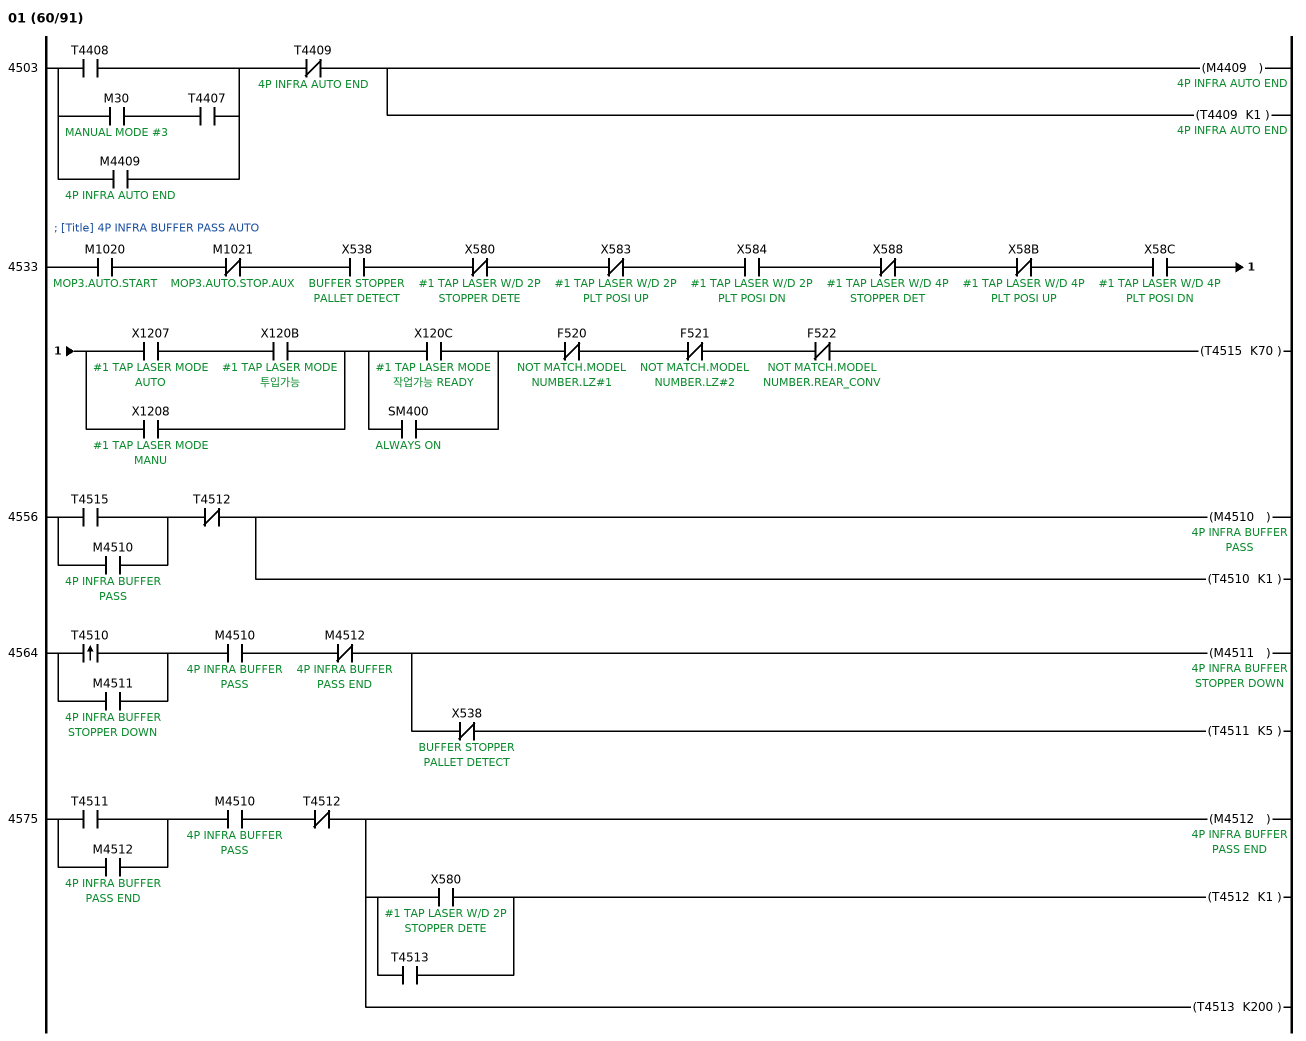
4503  LD      T4408
      LD      M30  ; MANUAL MODE #3
      AND     T4407
      ORB
      OR      M4409  ; 4P INFRA AUTO END
      ANI     T4409  ; 4P INFRA AUTO END
      OUT     M4409  ; 4P INFRA AUTO END
      OUT     T4409 K1  ; 4P INFRA AUTO END
; [Title] 4P INFRA BUFFER PASS AUTO
4533  LD      M1020  ; MOP3.AUTO.START
      ANI     M1021  ; MOP3.AUTO.STOP.AUX
      AND     X538  ; BUFFER STOPPER PALLET DETECT
      ANI     X580  ; #1 TAP LASER W/D 2P STOPPER DETE
      ANI     X583  ; #1 TAP LASER W/D 2P PLT POSI UP
      AND     X584  ; #1 TAP LASER W/D 2P PLT POSI DN
      ANI     X588  ; #1 TAP LASER W/D 4P STOPPER DET
      ANI     X58B  ; #1 TAP LASER W/D 4P PLT POSI UP
      AND     X58C  ; #1 TAP LASER W/D 4P PLT POSI DN
      LD      X1207  ; #1 TAP LASER MODE AUTO
      AND     X120B  ; #1 TAP LASER MODE 투입가능
      OR      X1208  ; #1 TAP LASER MODE MANU
      ANB
      LD      X120C  ; #1 TAP LASER MODE 작업가능 READY
      OR      SM400  ; ALWAYS ON
      ANB
      ANI     F520  ; NOT MATCH.MODEL NUMBER.LZ#1
      ANI     F521  ; NOT MATCH.MODEL NUMBER.LZ#2
      ANI     F522  ; NOT MATCH.MODEL NUMBER.REAR_CONV
      OUT     T4515 K70
4556  LD      T4515
      OR      M4510  ; 4P INFRA BUFFER PASS
      ANI     T4512
      OUT     M4510  ; 4P INFRA BUFFER PASS
      OUT     T4510 K1
4564  LDP     T4510
      OR      M4511  ; 4P INFRA BUFFER STOPPER DOWN
      AND     M4510  ; 4P INFRA BUFFER PASS
      ANI     M4512  ; 4P INFRA BUFFER PASS END
      OUT     M4511  ; 4P INFRA BUFFER STOPPER DOWN
      ANI     X538  ; BUFFER STOPPER PALLET DETECT
      OUT     T4511 K5
4575  LD      T4511
      OR      M4512  ; 4P INFRA BUFFER PASS END
      AND     M4510  ; 4P INFRA BUFFER PASS
      ANI     T4512
      OUT     M4512  ; 4P INFRA BUFFER PASS END
      MPS
      LD      X580  ; #1 TAP LASER W/D 2P STOPPER DETE
      OR      T4513
      ANB
      OUT     T4512 K1
      MPP
      OUT     T4513 K200
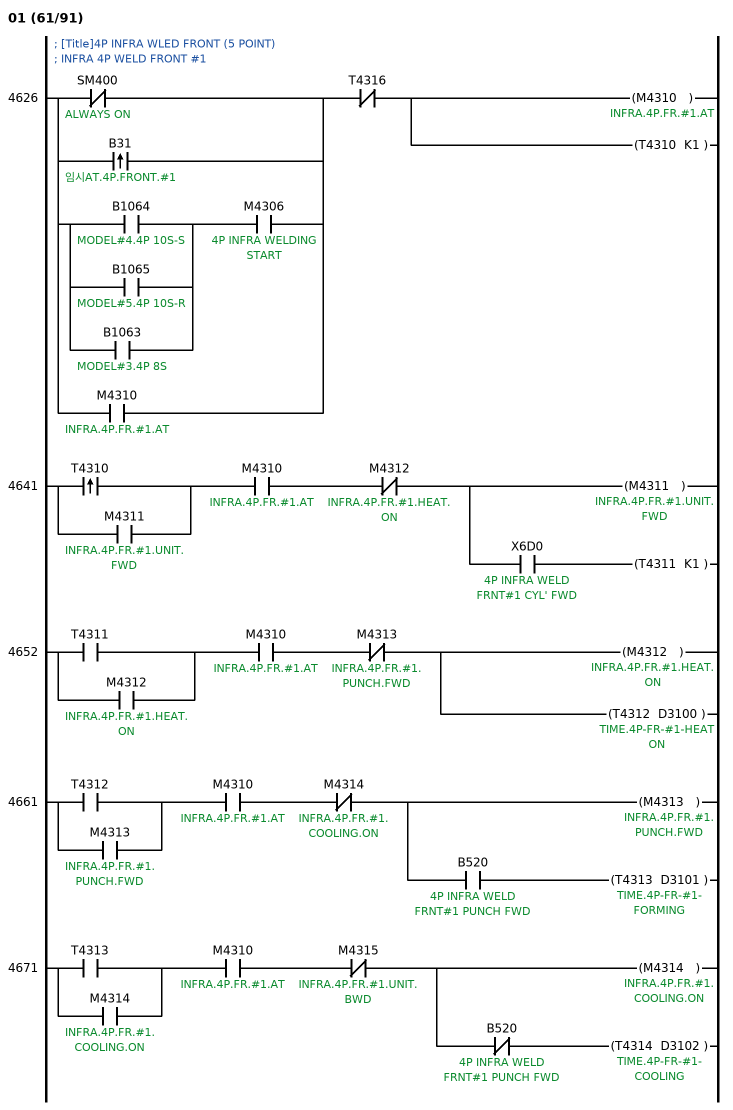
; [Title]4P INFRA WLED FRONT (5 POINT)
; INFRA 4P WELD FRONT #1
4626  LDI     SM400  ; ALWAYS ON
      ORP     B31  ; 임시AT.4P.FRONT.#1
      LD      B1064  ; MODEL#4.4P 10S-S
      OR      B1065  ; MODEL#5.4P 10S-R
      OR      B1063  ; MODEL#3.4P 8S
      AND     M4306  ; 4P INFRA WELDING START
      ORB
      OR      M4310  ; INFRA.4P.FR.#1.AT
      ANI     T4316
      OUT     M4310  ; INFRA.4P.FR.#1.AT
      OUT     T4310 K1
4641  LDP     T4310
      OR      M4311  ; INFRA.4P.FR.#1.UNIT.FWD
      AND     M4310  ; INFRA.4P.FR.#1.AT
      ANI     M4312  ; INFRA.4P.FR.#1.HEAT.ON
      OUT     M4311  ; INFRA.4P.FR.#1.UNIT.FWD
      AND     X6D0  ; 4P INFRA WELD FRNT#1 CYL' FWD
      OUT     T4311 K1
4652  LD      T4311
      OR      M4312  ; INFRA.4P.FR.#1.HEAT.ON
      AND     M4310  ; INFRA.4P.FR.#1.AT
      ANI     M4313  ; INFRA.4P.FR.#1.PUNCH.FWD
      OUT     M4312  ; INFRA.4P.FR.#1.HEAT.ON
      OUT     T4312 D3100  ; TIME.4P-FR-#1-HEAT ON
4661  LD      T4312
      OR      M4313  ; INFRA.4P.FR.#1.PUNCH.FWD
      AND     M4310  ; INFRA.4P.FR.#1.AT
      ANI     M4314  ; INFRA.4P.FR.#1.COOLING.ON
      OUT     M4313  ; INFRA.4P.FR.#1.PUNCH.FWD
      AND     B520  ; 4P INFRA WELD FRNT#1 PUNCH FWD
      OUT     T4313 D3101  ; TIME.4P-FR-#1-FORMING
4671  LD      T4313
      OR      M4314  ; INFRA.4P.FR.#1.COOLING.ON
      AND     M4310  ; INFRA.4P.FR.#1.AT
      ANI     M4315  ; INFRA.4P.FR.#1.UNIT.BWD
      OUT     M4314  ; INFRA.4P.FR.#1.COOLING.ON
      ANI     B520  ; 4P INFRA WELD FRNT#1 PUNCH FWD
      OUT     T4314 D3102  ; TIME.4P-FR-#1-COOLING
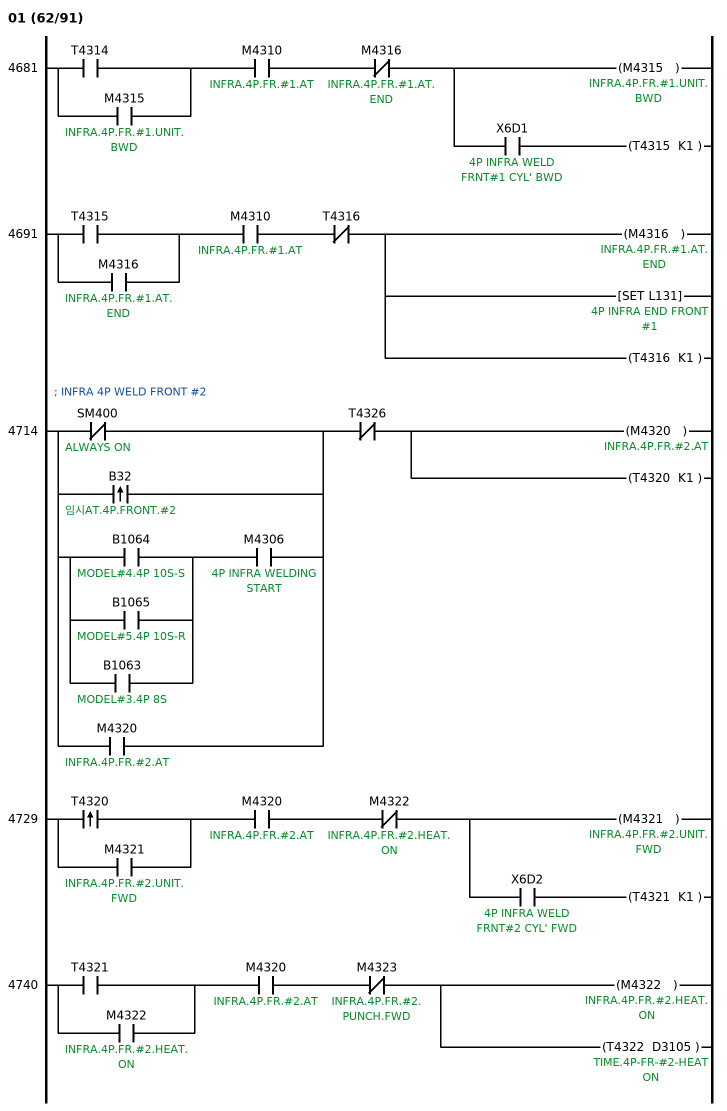
4681  LD      T4314
      OR      M4315  ; INFRA.4P.FR.#1.UNIT.BWD
      AND     M4310  ; INFRA.4P.FR.#1.AT
      ANI     M4316  ; INFRA.4P.FR.#1.AT.END
      OUT     M4315  ; INFRA.4P.FR.#1.UNIT.BWD
      AND     X6D1  ; 4P INFRA WELD FRNT#1 CYL' BWD
      OUT     T4315 K1
4691  LD      T4315
      OR      M4316  ; INFRA.4P.FR.#1.AT.END
      AND     M4310  ; INFRA.4P.FR.#1.AT
      ANI     T4316
      OUT     M4316  ; INFRA.4P.FR.#1.AT.END
      SET     L131  ; 4P INFRA END FRONT #1
      OUT     T4316 K1
; INFRA 4P WELD FRONT #2
4714  LDI     SM400  ; ALWAYS ON
      ORP     B32  ; 임시AT.4P.FRONT.#2
      LD      B1064  ; MODEL#4.4P 10S-S
      OR      B1065  ; MODEL#5.4P 10S-R
      OR      B1063  ; MODEL#3.4P 8S
      AND     M4306  ; 4P INFRA WELDING START
      ORB
      OR      M4320  ; INFRA.4P.FR.#2.AT
      ANI     T4326
      OUT     M4320  ; INFRA.4P.FR.#2.AT
      OUT     T4320 K1
4729  LDP     T4320
      OR      M4321  ; INFRA.4P.FR.#2.UNIT.FWD
      AND     M4320  ; INFRA.4P.FR.#2.AT
      ANI     M4322  ; INFRA.4P.FR.#2.HEAT.ON
      OUT     M4321  ; INFRA.4P.FR.#2.UNIT.FWD
      AND     X6D2  ; 4P INFRA WELD FRNT#2 CYL' FWD
      OUT     T4321 K1
4740  LD      T4321
      OR      M4322  ; INFRA.4P.FR.#2.HEAT.ON
      AND     M4320  ; INFRA.4P.FR.#2.AT
      ANI     M4323  ; INFRA.4P.FR.#2.PUNCH.FWD
      OUT     M4322  ; INFRA.4P.FR.#2.HEAT.ON
      OUT     T4322 D3105  ; TIME.4P-FR-#2-HEAT ON
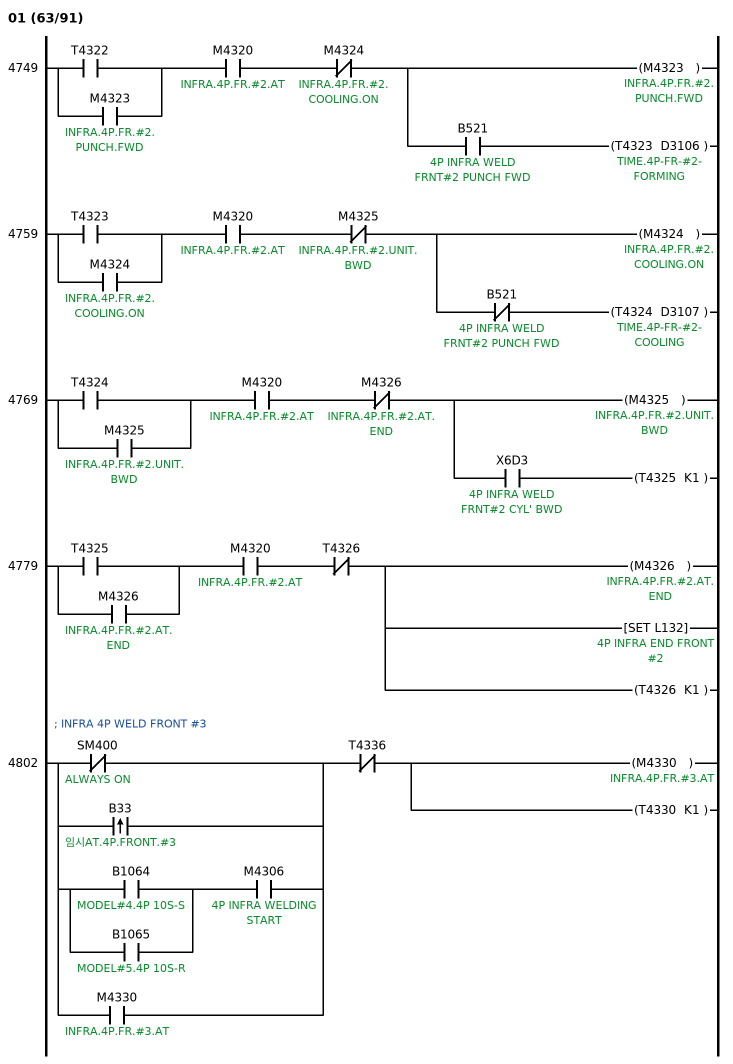
4749  LD      T4322
      OR      M4323  ; INFRA.4P.FR.#2.PUNCH.FWD
      AND     M4320  ; INFRA.4P.FR.#2.AT
      ANI     M4324  ; INFRA.4P.FR.#2.COOLING.ON
      OUT     M4323  ; INFRA.4P.FR.#2.PUNCH.FWD
      AND     B521  ; 4P INFRA WELD FRNT#2 PUNCH FWD
      OUT     T4323 D3106  ; TIME.4P-FR-#2-FORMING
4759  LD      T4323
      OR      M4324  ; INFRA.4P.FR.#2.COOLING.ON
      AND     M4320  ; INFRA.4P.FR.#2.AT
      ANI     M4325  ; INFRA.4P.FR.#2.UNIT.BWD
      OUT     M4324  ; INFRA.4P.FR.#2.COOLING.ON
      ANI     B521  ; 4P INFRA WELD FRNT#2 PUNCH FWD
      OUT     T4324 D3107  ; TIME.4P-FR-#2-COOLING
4769  LD      T4324
      OR      M4325  ; INFRA.4P.FR.#2.UNIT.BWD
      AND     M4320  ; INFRA.4P.FR.#2.AT
      ANI     M4326  ; INFRA.4P.FR.#2.AT.END
      OUT     M4325  ; INFRA.4P.FR.#2.UNIT.BWD
      AND     X6D3  ; 4P INFRA WELD FRNT#2 CYL' BWD
      OUT     T4325 K1
4779  LD      T4325
      OR      M4326  ; INFRA.4P.FR.#2.AT.END
      AND     M4320  ; INFRA.4P.FR.#2.AT
      ANI     T4326
      OUT     M4326  ; INFRA.4P.FR.#2.AT.END
      SET     L132  ; 4P INFRA END FRONT #2
      OUT     T4326 K1
; INFRA 4P WELD FRONT #3
4802  LDI     SM400  ; ALWAYS ON
      ORP     B33  ; 임시AT.4P.FRONT.#3
      LD      B1064  ; MODEL#4.4P 10S-S
      OR      B1065  ; MODEL#5.4P 10S-R
      AND     M4306  ; 4P INFRA WELDING START
      ORB
      OR      M4330  ; INFRA.4P.FR.#3.AT
      ANI     T4336
      OUT     M4330  ; INFRA.4P.FR.#3.AT
      OUT     T4330 K1
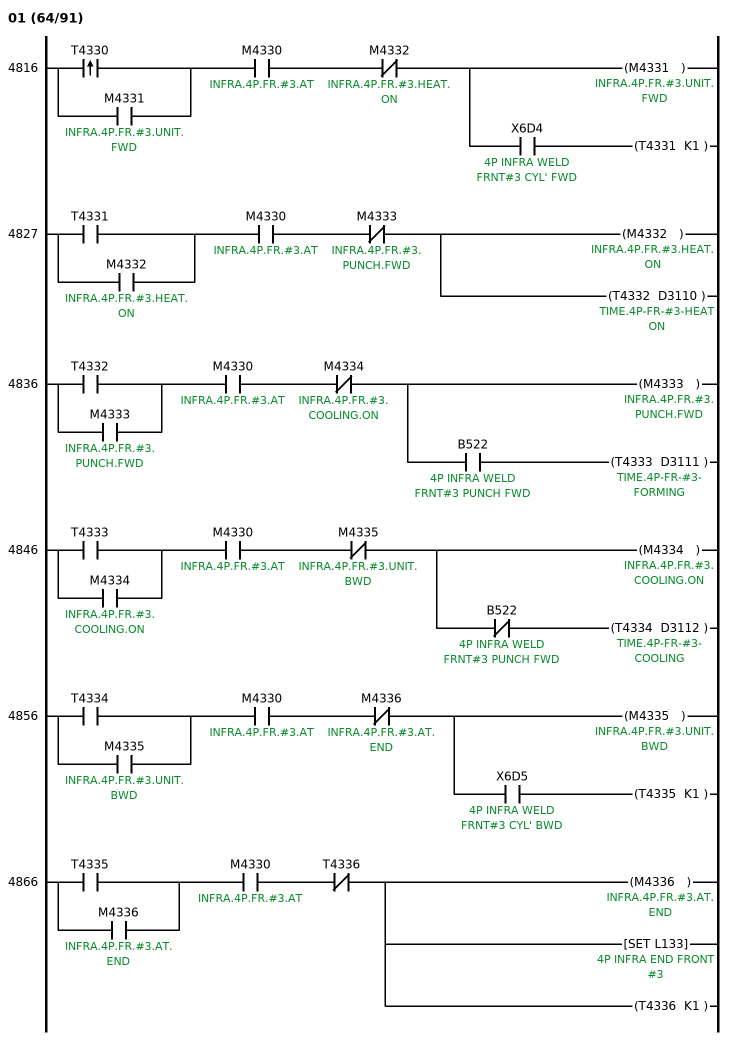
4816  LDP     T4330
      OR      M4331  ; INFRA.4P.FR.#3.UNIT.FWD
      AND     M4330  ; INFRA.4P.FR.#3.AT
      ANI     M4332  ; INFRA.4P.FR.#3.HEAT.ON
      OUT     M4331  ; INFRA.4P.FR.#3.UNIT.FWD
      AND     X6D4  ; 4P INFRA WELD FRNT#3 CYL' FWD
      OUT     T4331 K1
4827  LD      T4331
      OR      M4332  ; INFRA.4P.FR.#3.HEAT.ON
      AND     M4330  ; INFRA.4P.FR.#3.AT
      ANI     M4333  ; INFRA.4P.FR.#3.PUNCH.FWD
      OUT     M4332  ; INFRA.4P.FR.#3.HEAT.ON
      OUT     T4332 D3110  ; TIME.4P-FR-#3-HEAT ON
4836  LD      T4332
      OR      M4333  ; INFRA.4P.FR.#3.PUNCH.FWD
      AND     M4330  ; INFRA.4P.FR.#3.AT
      ANI     M4334  ; INFRA.4P.FR.#3.COOLING.ON
      OUT     M4333  ; INFRA.4P.FR.#3.PUNCH.FWD
      AND     B522  ; 4P INFRA WELD FRNT#3 PUNCH FWD
      OUT     T4333 D3111  ; TIME.4P-FR-#3-FORMING
4846  LD      T4333
      OR      M4334  ; INFRA.4P.FR.#3.COOLING.ON
      AND     M4330  ; INFRA.4P.FR.#3.AT
      ANI     M4335  ; INFRA.4P.FR.#3.UNIT.BWD
      OUT     M4334  ; INFRA.4P.FR.#3.COOLING.ON
      ANI     B522  ; 4P INFRA WELD FRNT#3 PUNCH FWD
      OUT     T4334 D3112  ; TIME.4P-FR-#3-COOLING
4856  LD      T4334
      OR      M4335  ; INFRA.4P.FR.#3.UNIT.BWD
      AND     M4330  ; INFRA.4P.FR.#3.AT
      ANI     M4336  ; INFRA.4P.FR.#3.AT.END
      OUT     M4335  ; INFRA.4P.FR.#3.UNIT.BWD
      AND     X6D5  ; 4P INFRA WELD FRNT#3 CYL' BWD
      OUT     T4335 K1
4866  LD      T4335
      OR      M4336  ; INFRA.4P.FR.#3.AT.END
      AND     M4330  ; INFRA.4P.FR.#3.AT
      ANI     T4336
      OUT     M4336  ; INFRA.4P.FR.#3.AT.END
      SET     L133  ; 4P INFRA END FRONT #3
      OUT     T4336 K1
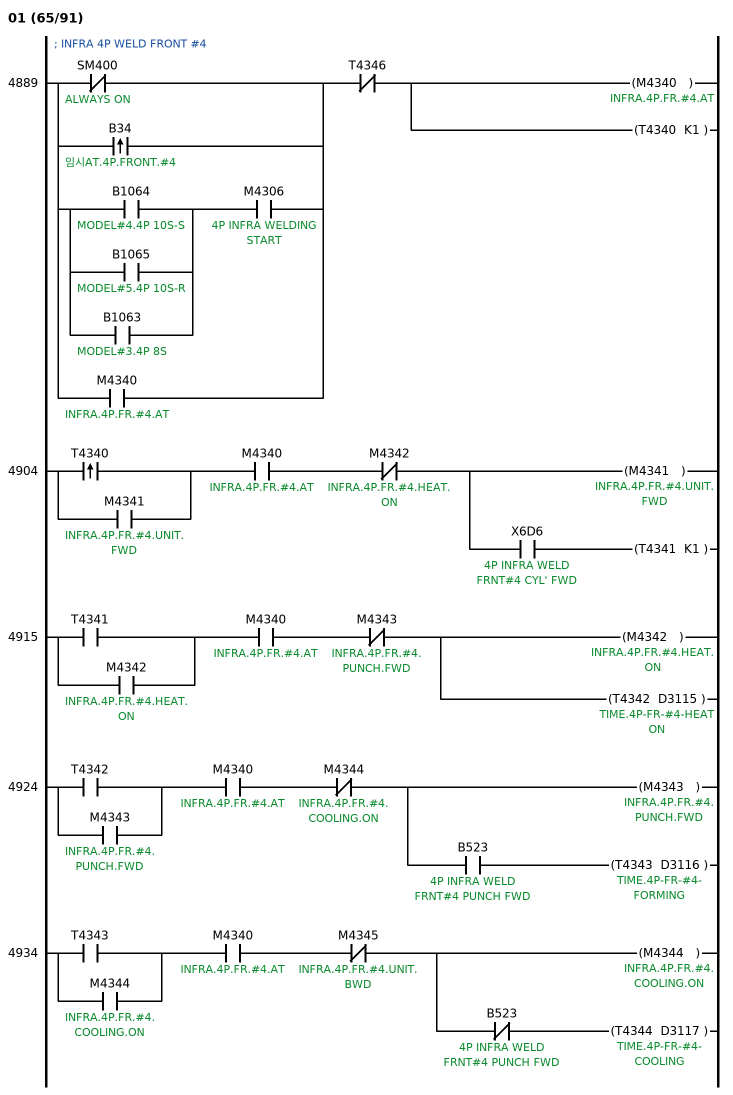
; INFRA 4P WELD FRONT #4
4889  LDI     SM400  ; ALWAYS ON
      ORP     B34  ; 임시AT.4P.FRONT.#4
      LD      B1064  ; MODEL#4.4P 10S-S
      OR      B1065  ; MODEL#5.4P 10S-R
      OR      B1063  ; MODEL#3.4P 8S
      AND     M4306  ; 4P INFRA WELDING START
      ORB
      OR      M4340  ; INFRA.4P.FR.#4.AT
      ANI     T4346
      OUT     M4340  ; INFRA.4P.FR.#4.AT
      OUT     T4340 K1
4904  LDP     T4340
      OR      M4341  ; INFRA.4P.FR.#4.UNIT.FWD
      AND     M4340  ; INFRA.4P.FR.#4.AT
      ANI     M4342  ; INFRA.4P.FR.#4.HEAT.ON
      OUT     M4341  ; INFRA.4P.FR.#4.UNIT.FWD
      AND     X6D6  ; 4P INFRA WELD FRNT#4 CYL' FWD
      OUT     T4341 K1
4915  LD      T4341
      OR      M4342  ; INFRA.4P.FR.#4.HEAT.ON
      AND     M4340  ; INFRA.4P.FR.#4.AT
      ANI     M4343  ; INFRA.4P.FR.#4.PUNCH.FWD
      OUT     M4342  ; INFRA.4P.FR.#4.HEAT.ON
      OUT     T4342 D3115  ; TIME.4P-FR-#4-HEAT ON
4924  LD      T4342
      OR      M4343  ; INFRA.4P.FR.#4.PUNCH.FWD
      AND     M4340  ; INFRA.4P.FR.#4.AT
      ANI     M4344  ; INFRA.4P.FR.#4.COOLING.ON
      OUT     M4343  ; INFRA.4P.FR.#4.PUNCH.FWD
      AND     B523  ; 4P INFRA WELD FRNT#4 PUNCH FWD
      OUT     T4343 D3116  ; TIME.4P-FR-#4-FORMING
4934  LD      T4343
      OR      M4344  ; INFRA.4P.FR.#4.COOLING.ON
      AND     M4340  ; INFRA.4P.FR.#4.AT
      ANI     M4345  ; INFRA.4P.FR.#4.UNIT.BWD
      OUT     M4344  ; INFRA.4P.FR.#4.COOLING.ON
      ANI     B523  ; 4P INFRA WELD FRNT#4 PUNCH FWD
      OUT     T4344 D3117  ; TIME.4P-FR-#4-COOLING
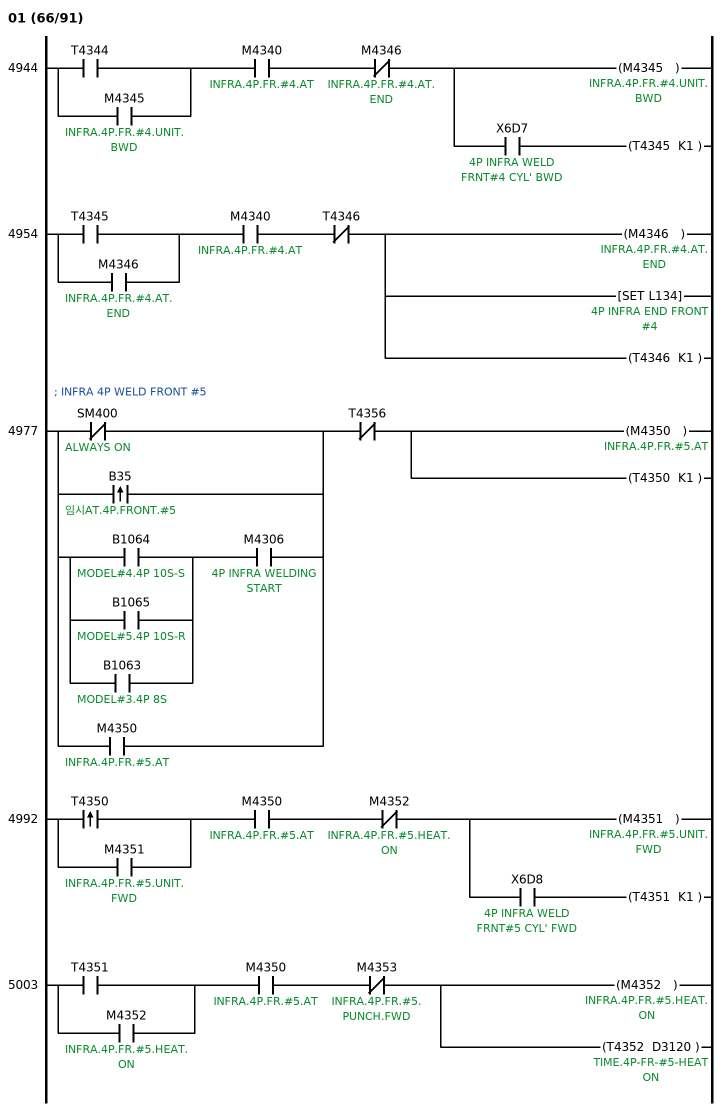
4944  LD      T4344
      OR      M4345  ; INFRA.4P.FR.#4.UNIT.BWD
      AND     M4340  ; INFRA.4P.FR.#4.AT
      ANI     M4346  ; INFRA.4P.FR.#4.AT.END
      OUT     M4345  ; INFRA.4P.FR.#4.UNIT.BWD
      AND     X6D7  ; 4P INFRA WELD FRNT#4 CYL' BWD
      OUT     T4345 K1
4954  LD      T4345
      OR      M4346  ; INFRA.4P.FR.#4.AT.END
      AND     M4340  ; INFRA.4P.FR.#4.AT
      ANI     T4346
      OUT     M4346  ; INFRA.4P.FR.#4.AT.END
      SET     L134  ; 4P INFRA END FRONT #4
      OUT     T4346 K1
; INFRA 4P WELD FRONT #5
4977  LDI     SM400  ; ALWAYS ON
      ORP     B35  ; 임시AT.4P.FRONT.#5
      LD      B1064  ; MODEL#4.4P 10S-S
      OR      B1065  ; MODEL#5.4P 10S-R
      OR      B1063  ; MODEL#3.4P 8S
      AND     M4306  ; 4P INFRA WELDING START
      ORB
      OR      M4350  ; INFRA.4P.FR.#5.AT
      ANI     T4356
      OUT     M4350  ; INFRA.4P.FR.#5.AT
      OUT     T4350 K1
4992  LDP     T4350
      OR      M4351  ; INFRA.4P.FR.#5.UNIT.FWD
      AND     M4350  ; INFRA.4P.FR.#5.AT
      ANI     M4352  ; INFRA.4P.FR.#5.HEAT.ON
      OUT     M4351  ; INFRA.4P.FR.#5.UNIT.FWD
      AND     X6D8  ; 4P INFRA WELD FRNT#5 CYL' FWD
      OUT     T4351 K1
5003  LD      T4351
      OR      M4352  ; INFRA.4P.FR.#5.HEAT.ON
      AND     M4350  ; INFRA.4P.FR.#5.AT
      ANI     M4353  ; INFRA.4P.FR.#5.PUNCH.FWD
      OUT     M4352  ; INFRA.4P.FR.#5.HEAT.ON
      OUT     T4352 D3120  ; TIME.4P-FR-#5-HEAT ON
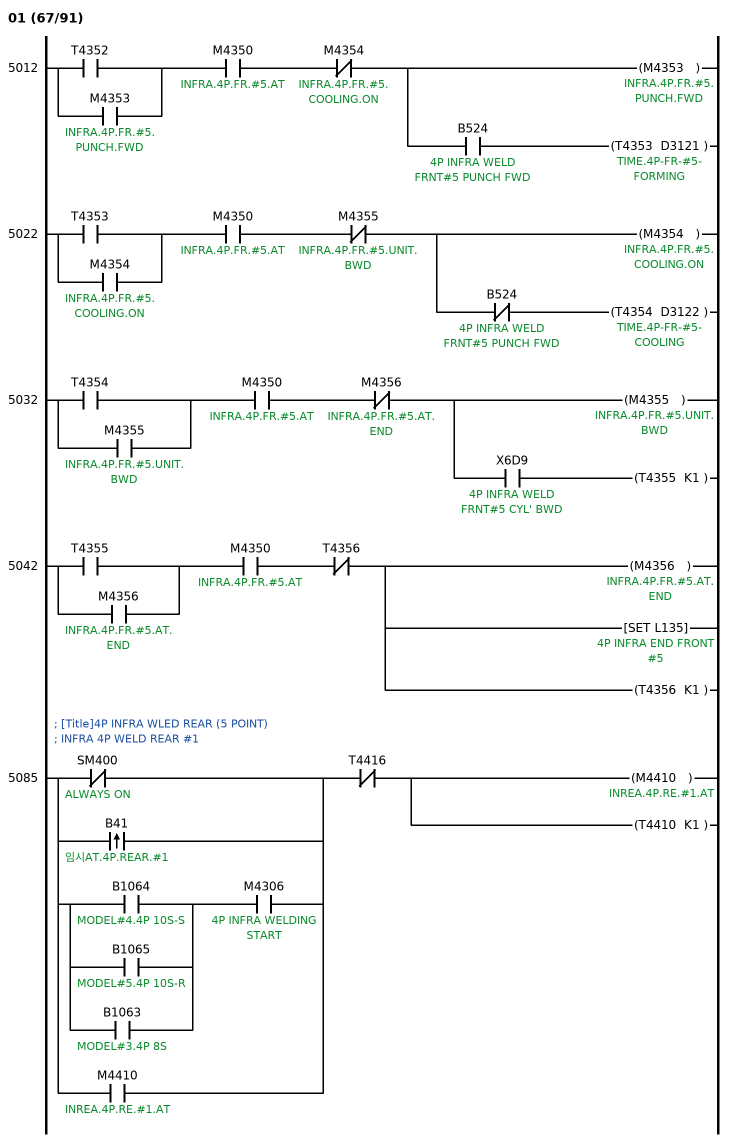
5012  LD      T4352
      OR      M4353  ; INFRA.4P.FR.#5.PUNCH.FWD
      AND     M4350  ; INFRA.4P.FR.#5.AT
      ANI     M4354  ; INFRA.4P.FR.#5.COOLING.ON
      OUT     M4353  ; INFRA.4P.FR.#5.PUNCH.FWD
      AND     B524  ; 4P INFRA WELD FRNT#5 PUNCH FWD
      OUT     T4353 D3121  ; TIME.4P-FR-#5-FORMING
5022  LD      T4353
      OR      M4354  ; INFRA.4P.FR.#5.COOLING.ON
      AND     M4350  ; INFRA.4P.FR.#5.AT
      ANI     M4355  ; INFRA.4P.FR.#5.UNIT.BWD
      OUT     M4354  ; INFRA.4P.FR.#5.COOLING.ON
      ANI     B524  ; 4P INFRA WELD FRNT#5 PUNCH FWD
      OUT     T4354 D3122  ; TIME.4P-FR-#5-COOLING
5032  LD      T4354
      OR      M4355  ; INFRA.4P.FR.#5.UNIT.BWD
      AND     M4350  ; INFRA.4P.FR.#5.AT
      ANI     M4356  ; INFRA.4P.FR.#5.AT.END
      OUT     M4355  ; INFRA.4P.FR.#5.UNIT.BWD
      AND     X6D9  ; 4P INFRA WELD FRNT#5 CYL' BWD
      OUT     T4355 K1
5042  LD      T4355
      OR      M4356  ; INFRA.4P.FR.#5.AT.END
      AND     M4350  ; INFRA.4P.FR.#5.AT
      ANI     T4356
      OUT     M4356  ; INFRA.4P.FR.#5.AT.END
      SET     L135  ; 4P INFRA END FRONT #5
      OUT     T4356 K1
; [Title]4P INFRA WLED REAR (5 POINT)
; INFRA 4P WELD REAR #1
5085  LDI     SM400  ; ALWAYS ON
      ORP     B41  ; 임시AT.4P.REAR.#1
      LD      B1064  ; MODEL#4.4P 10S-S
      OR      B1065  ; MODEL#5.4P 10S-R
      OR      B1063  ; MODEL#3.4P 8S
      AND     M4306  ; 4P INFRA WELDING START
      ORB
      OR      M4410  ; INREA.4P.RE.#1.AT
      ANI     T4416
      OUT     M4410  ; INREA.4P.RE.#1.AT
      OUT     T4410 K1
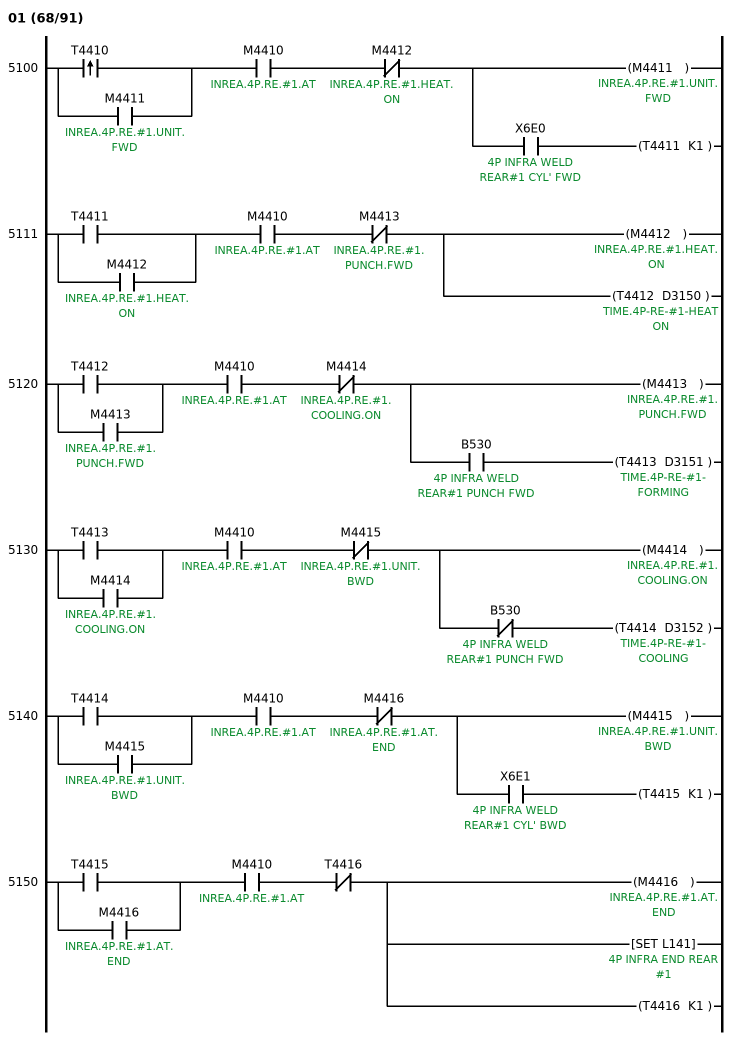
5100  LDP     T4410
      OR      M4411  ; INREA.4P.RE.#1.UNIT.FWD
      AND     M4410  ; INREA.4P.RE.#1.AT
      ANI     M4412  ; INREA.4P.RE.#1.HEAT.ON
      OUT     M4411  ; INREA.4P.RE.#1.UNIT.FWD
      AND     X6E0  ; 4P INFRA WELD REAR#1 CYL' FWD
      OUT     T4411 K1
5111  LD      T4411
      OR      M4412  ; INREA.4P.RE.#1.HEAT.ON
      AND     M4410  ; INREA.4P.RE.#1.AT
      ANI     M4413  ; INREA.4P.RE.#1.PUNCH.FWD
      OUT     M4412  ; INREA.4P.RE.#1.HEAT.ON
      OUT     T4412 D3150  ; TIME.4P-RE-#1-HEAT ON
5120  LD      T4412
      OR      M4413  ; INREA.4P.RE.#1.PUNCH.FWD
      AND     M4410  ; INREA.4P.RE.#1.AT
      ANI     M4414  ; INREA.4P.RE.#1.COOLING.ON
      OUT     M4413  ; INREA.4P.RE.#1.PUNCH.FWD
      AND     B530  ; 4P INFRA WELD REAR#1 PUNCH FWD
      OUT     T4413 D3151  ; TIME.4P-RE-#1-FORMING
5130  LD      T4413
      OR      M4414  ; INREA.4P.RE.#1.COOLING.ON
      AND     M4410  ; INREA.4P.RE.#1.AT
      ANI     M4415  ; INREA.4P.RE.#1.UNIT.BWD
      OUT     M4414  ; INREA.4P.RE.#1.COOLING.ON
      ANI     B530  ; 4P INFRA WELD REAR#1 PUNCH FWD
      OUT     T4414 D3152  ; TIME.4P-RE-#1-COOLING
5140  LD      T4414
      OR      M4415  ; INREA.4P.RE.#1.UNIT.BWD
      AND     M4410  ; INREA.4P.RE.#1.AT
      ANI     M4416  ; INREA.4P.RE.#1.AT.END
      OUT     M4415  ; INREA.4P.RE.#1.UNIT.BWD
      AND     X6E1  ; 4P INFRA WELD REAR#1 CYL' BWD
      OUT     T4415 K1
5150  LD      T4415
      OR      M4416  ; INREA.4P.RE.#1.AT.END
      AND     M4410  ; INREA.4P.RE.#1.AT
      ANI     T4416
      OUT     M4416  ; INREA.4P.RE.#1.AT.END
      SET     L141  ; 4P INFRA END REAR #1
      OUT     T4416 K1
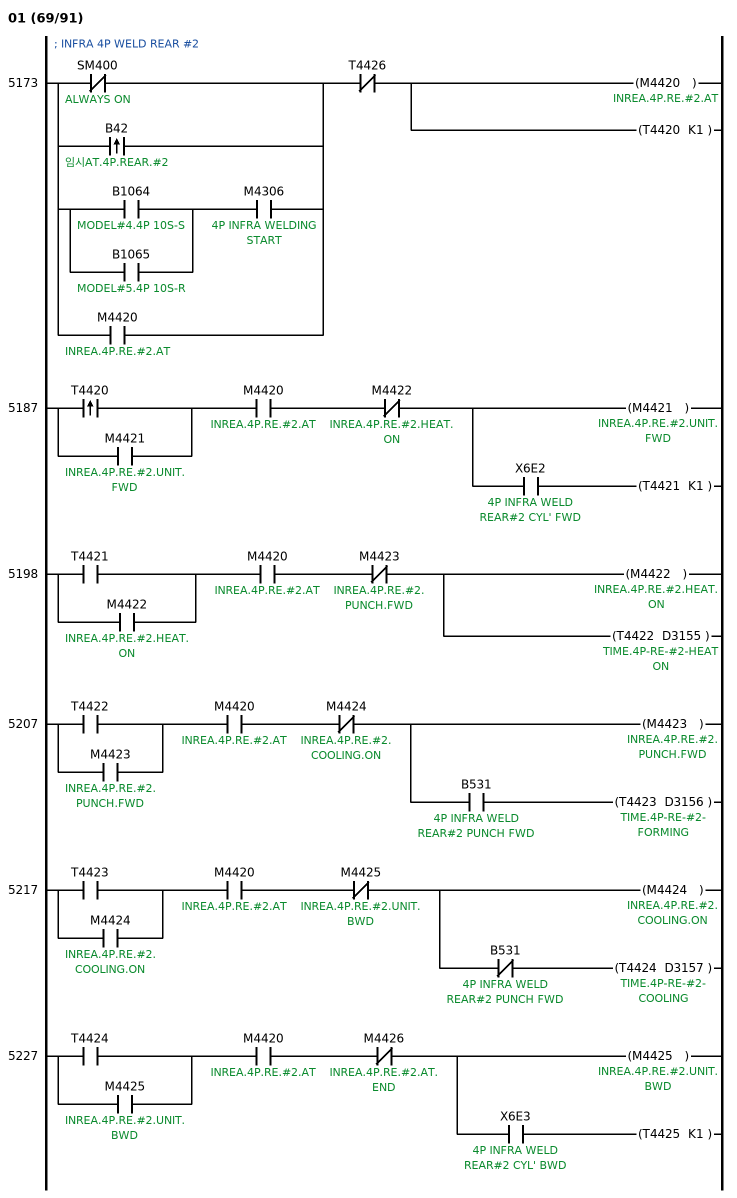
; INFRA 4P WELD REAR #2
5173  LDI     SM400  ; ALWAYS ON
      ORP     B42  ; 임시AT.4P.REAR.#2
      LD      B1064  ; MODEL#4.4P 10S-S
      OR      B1065  ; MODEL#5.4P 10S-R
      AND     M4306  ; 4P INFRA WELDING START
      ORB
      OR      M4420  ; INREA.4P.RE.#2.AT
      ANI     T4426
      OUT     M4420  ; INREA.4P.RE.#2.AT
      OUT     T4420 K1
5187  LDP     T4420
      OR      M4421  ; INREA.4P.RE.#2.UNIT.FWD
      AND     M4420  ; INREA.4P.RE.#2.AT
      ANI     M4422  ; INREA.4P.RE.#2.HEAT.ON
      OUT     M4421  ; INREA.4P.RE.#2.UNIT.FWD
      AND     X6E2  ; 4P INFRA WELD REAR#2 CYL' FWD
      OUT     T4421 K1
5198  LD      T4421
      OR      M4422  ; INREA.4P.RE.#2.HEAT.ON
      AND     M4420  ; INREA.4P.RE.#2.AT
      ANI     M4423  ; INREA.4P.RE.#2.PUNCH.FWD
      OUT     M4422  ; INREA.4P.RE.#2.HEAT.ON
      OUT     T4422 D3155  ; TIME.4P-RE-#2-HEAT ON
5207  LD      T4422
      OR      M4423  ; INREA.4P.RE.#2.PUNCH.FWD
      AND     M4420  ; INREA.4P.RE.#2.AT
      ANI     M4424  ; INREA.4P.RE.#2.COOLING.ON
      OUT     M4423  ; INREA.4P.RE.#2.PUNCH.FWD
      AND     B531  ; 4P INFRA WELD REAR#2 PUNCH FWD
      OUT     T4423 D3156  ; TIME.4P-RE-#2-FORMING
5217  LD      T4423
      OR      M4424  ; INREA.4P.RE.#2.COOLING.ON
      AND     M4420  ; INREA.4P.RE.#2.AT
      ANI     M4425  ; INREA.4P.RE.#2.UNIT.BWD
      OUT     M4424  ; INREA.4P.RE.#2.COOLING.ON
      ANI     B531  ; 4P INFRA WELD REAR#2 PUNCH FWD
      OUT     T4424 D3157  ; TIME.4P-RE-#2-COOLING
5227  LD      T4424
      OR      M4425  ; INREA.4P.RE.#2.UNIT.BWD
      AND     M4420  ; INREA.4P.RE.#2.AT
      ANI     M4426  ; INREA.4P.RE.#2.AT.END
      OUT     M4425  ; INREA.4P.RE.#2.UNIT.BWD
      AND     X6E3  ; 4P INFRA WELD REAR#2 CYL' BWD
      OUT     T4425 K1
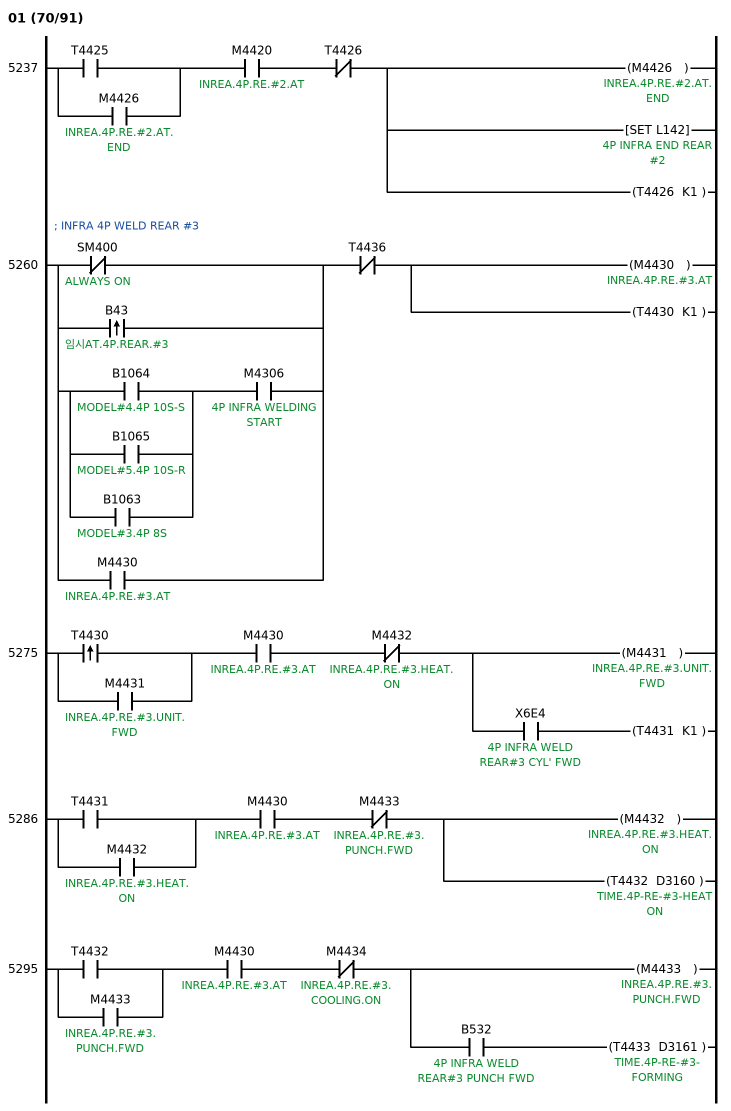
5237  LD      T4425
      OR      M4426  ; INREA.4P.RE.#2.AT.END
      AND     M4420  ; INREA.4P.RE.#2.AT
      ANI     T4426
      OUT     M4426  ; INREA.4P.RE.#2.AT.END
      SET     L142  ; 4P INFRA END REAR #2
      OUT     T4426 K1
; INFRA 4P WELD REAR #3
5260  LDI     SM400  ; ALWAYS ON
      ORP     B43  ; 임시AT.4P.REAR.#3
      LD      B1064  ; MODEL#4.4P 10S-S
      OR      B1065  ; MODEL#5.4P 10S-R
      OR      B1063  ; MODEL#3.4P 8S
      AND     M4306  ; 4P INFRA WELDING START
      ORB
      OR      M4430  ; INREA.4P.RE.#3.AT
      ANI     T4436
      OUT     M4430  ; INREA.4P.RE.#3.AT
      OUT     T4430 K1
5275  LDP     T4430
      OR      M4431  ; INREA.4P.RE.#3.UNIT.FWD
      AND     M4430  ; INREA.4P.RE.#3.AT
      ANI     M4432  ; INREA.4P.RE.#3.HEAT.ON
      OUT     M4431  ; INREA.4P.RE.#3.UNIT.FWD
      AND     X6E4  ; 4P INFRA WELD REAR#3 CYL' FWD
      OUT     T4431 K1
5286  LD      T4431
      OR      M4432  ; INREA.4P.RE.#3.HEAT.ON
      AND     M4430  ; INREA.4P.RE.#3.AT
      ANI     M4433  ; INREA.4P.RE.#3.PUNCH.FWD
      OUT     M4432  ; INREA.4P.RE.#3.HEAT.ON
      OUT     T4432 D3160  ; TIME.4P-RE-#3-HEAT ON
5295  LD      T4432
      OR      M4433  ; INREA.4P.RE.#3.PUNCH.FWD
      AND     M4430  ; INREA.4P.RE.#3.AT
      ANI     M4434  ; INREA.4P.RE.#3.COOLING.ON
      OUT     M4433  ; INREA.4P.RE.#3.PUNCH.FWD
      AND     B532  ; 4P INFRA WELD REAR#3 PUNCH FWD
      OUT     T4433 D3161  ; TIME.4P-RE-#3-FORMING
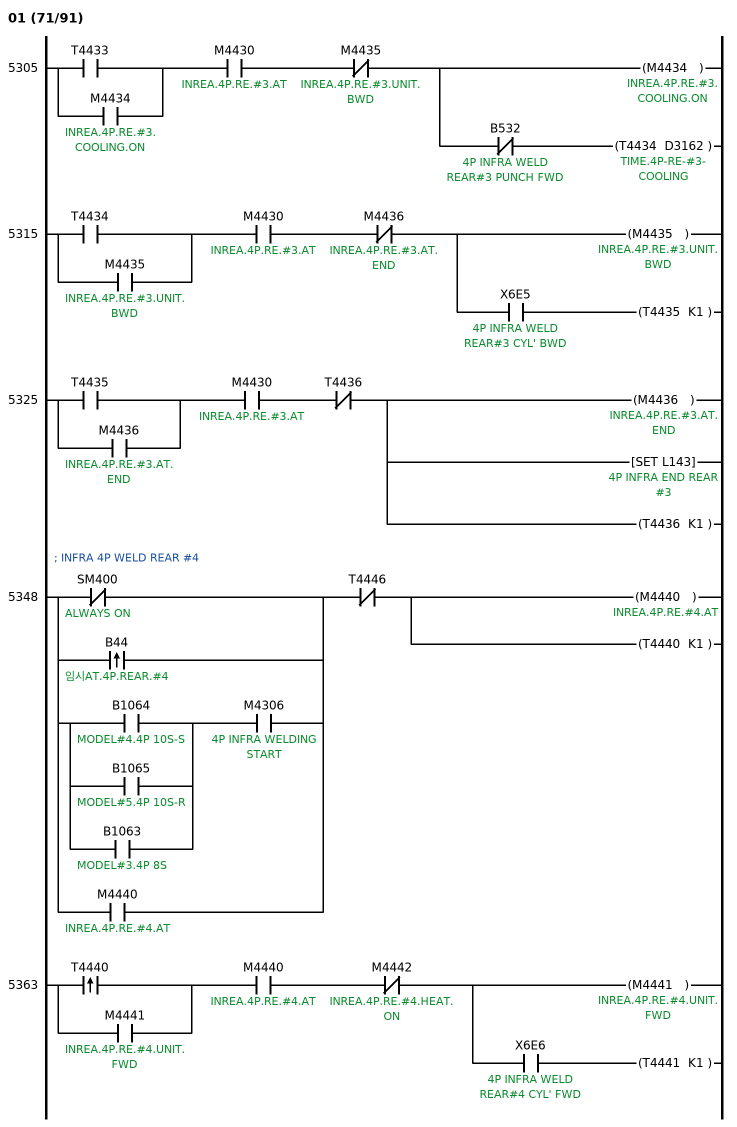
5305  LD      T4433
      OR      M4434  ; INREA.4P.RE.#3.COOLING.ON
      AND     M4430  ; INREA.4P.RE.#3.AT
      ANI     M4435  ; INREA.4P.RE.#3.UNIT.BWD
      OUT     M4434  ; INREA.4P.RE.#3.COOLING.ON
      ANI     B532  ; 4P INFRA WELD REAR#3 PUNCH FWD
      OUT     T4434 D3162  ; TIME.4P-RE-#3-COOLING
5315  LD      T4434
      OR      M4435  ; INREA.4P.RE.#3.UNIT.BWD
      AND     M4430  ; INREA.4P.RE.#3.AT
      ANI     M4436  ; INREA.4P.RE.#3.AT.END
      OUT     M4435  ; INREA.4P.RE.#3.UNIT.BWD
      AND     X6E5  ; 4P INFRA WELD REAR#3 CYL' BWD
      OUT     T4435 K1
5325  LD      T4435
      OR      M4436  ; INREA.4P.RE.#3.AT.END
      AND     M4430  ; INREA.4P.RE.#3.AT
      ANI     T4436
      OUT     M4436  ; INREA.4P.RE.#3.AT.END
      SET     L143  ; 4P INFRA END REAR #3
      OUT     T4436 K1
; INFRA 4P WELD REAR #4
5348  LDI     SM400  ; ALWAYS ON
      ORP     B44  ; 임시AT.4P.REAR.#4
      LD      B1064  ; MODEL#4.4P 10S-S
      OR      B1065  ; MODEL#5.4P 10S-R
      OR      B1063  ; MODEL#3.4P 8S
      AND     M4306  ; 4P INFRA WELDING START
      ORB
      OR      M4440  ; INREA.4P.RE.#4.AT
      ANI     T4446
      OUT     M4440  ; INREA.4P.RE.#4.AT
      OUT     T4440 K1
5363  LDP     T4440
      OR      M4441  ; INREA.4P.RE.#4.UNIT.FWD
      AND     M4440  ; INREA.4P.RE.#4.AT
      ANI     M4442  ; INREA.4P.RE.#4.HEAT.ON
      OUT     M4441  ; INREA.4P.RE.#4.UNIT.FWD
      AND     X6E6  ; 4P INFRA WELD REAR#4 CYL' FWD
      OUT     T4441 K1
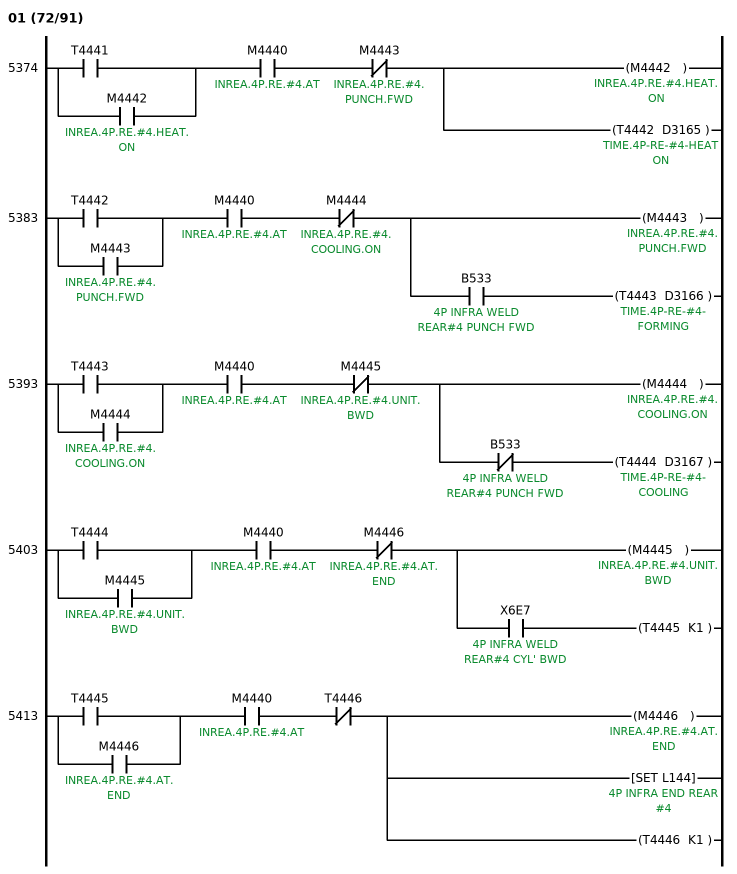
5374  LD      T4441
      OR      M4442  ; INREA.4P.RE.#4.HEAT.ON
      AND     M4440  ; INREA.4P.RE.#4.AT
      ANI     M4443  ; INREA.4P.RE.#4.PUNCH.FWD
      OUT     M4442  ; INREA.4P.RE.#4.HEAT.ON
      OUT     T4442 D3165  ; TIME.4P-RE-#4-HEAT ON
5383  LD      T4442
      OR      M4443  ; INREA.4P.RE.#4.PUNCH.FWD
      AND     M4440  ; INREA.4P.RE.#4.AT
      ANI     M4444  ; INREA.4P.RE.#4.COOLING.ON
      OUT     M4443  ; INREA.4P.RE.#4.PUNCH.FWD
      AND     B533  ; 4P INFRA WELD REAR#4 PUNCH FWD
      OUT     T4443 D3166  ; TIME.4P-RE-#4-FORMING
5393  LD      T4443
      OR      M4444  ; INREA.4P.RE.#4.COOLING.ON
      AND     M4440  ; INREA.4P.RE.#4.AT
      ANI     M4445  ; INREA.4P.RE.#4.UNIT.BWD
      OUT     M4444  ; INREA.4P.RE.#4.COOLING.ON
      ANI     B533  ; 4P INFRA WELD REAR#4 PUNCH FWD
      OUT     T4444 D3167  ; TIME.4P-RE-#4-COOLING
5403  LD      T4444
      OR      M4445  ; INREA.4P.RE.#4.UNIT.BWD
      AND     M4440  ; INREA.4P.RE.#4.AT
      ANI     M4446  ; INREA.4P.RE.#4.AT.END
      OUT     M4445  ; INREA.4P.RE.#4.UNIT.BWD
      AND     X6E7  ; 4P INFRA WELD REAR#4 CYL' BWD
      OUT     T4445 K1
5413  LD      T4445
      OR      M4446  ; INREA.4P.RE.#4.AT.END
      AND     M4440  ; INREA.4P.RE.#4.AT
      ANI     T4446
      OUT     M4446  ; INREA.4P.RE.#4.AT.END
      SET     L144  ; 4P INFRA END REAR #4
      OUT     T4446 K1
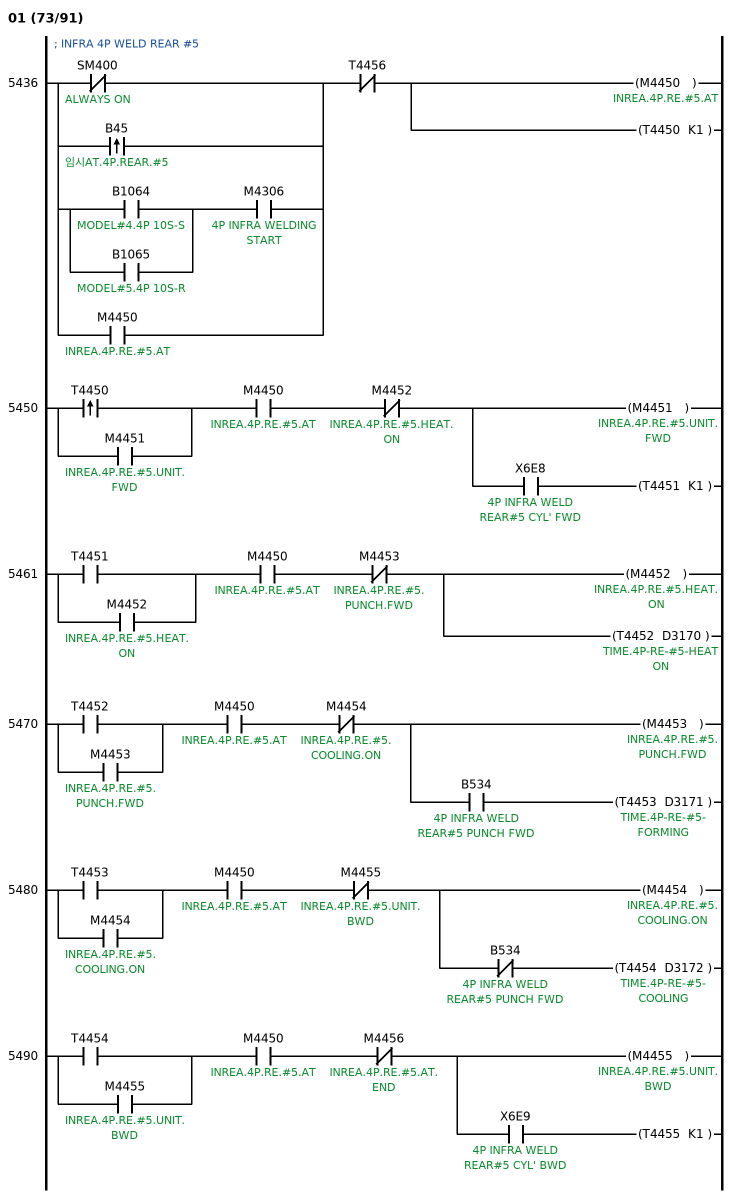
; INFRA 4P WELD REAR #5
5436  LDI     SM400  ; ALWAYS ON
      ORP     B45  ; 임시AT.4P.REAR.#5
      LD      B1064  ; MODEL#4.4P 10S-S
      OR      B1065  ; MODEL#5.4P 10S-R
      AND     M4306  ; 4P INFRA WELDING START
      ORB
      OR      M4450  ; INREA.4P.RE.#5.AT
      ANI     T4456
      OUT     M4450  ; INREA.4P.RE.#5.AT
      OUT     T4450 K1
5450  LDP     T4450
      OR      M4451  ; INREA.4P.RE.#5.UNIT.FWD
      AND     M4450  ; INREA.4P.RE.#5.AT
      ANI     M4452  ; INREA.4P.RE.#5.HEAT.ON
      OUT     M4451  ; INREA.4P.RE.#5.UNIT.FWD
      AND     X6E8  ; 4P INFRA WELD REAR#5 CYL' FWD
      OUT     T4451 K1
5461  LD      T4451
      OR      M4452  ; INREA.4P.RE.#5.HEAT.ON
      AND     M4450  ; INREA.4P.RE.#5.AT
      ANI     M4453  ; INREA.4P.RE.#5.PUNCH.FWD
      OUT     M4452  ; INREA.4P.RE.#5.HEAT.ON
      OUT     T4452 D3170  ; TIME.4P-RE-#5-HEAT ON
5470  LD      T4452
      OR      M4453  ; INREA.4P.RE.#5.PUNCH.FWD
      AND     M4450  ; INREA.4P.RE.#5.AT
      ANI     M4454  ; INREA.4P.RE.#5.COOLING.ON
      OUT     M4453  ; INREA.4P.RE.#5.PUNCH.FWD
      AND     B534  ; 4P INFRA WELD REAR#5 PUNCH FWD
      OUT     T4453 D3171  ; TIME.4P-RE-#5-FORMING
5480  LD      T4453
      OR      M4454  ; INREA.4P.RE.#5.COOLING.ON
      AND     M4450  ; INREA.4P.RE.#5.AT
      ANI     M4455  ; INREA.4P.RE.#5.UNIT.BWD
      OUT     M4454  ; INREA.4P.RE.#5.COOLING.ON
      ANI     B534  ; 4P INFRA WELD REAR#5 PUNCH FWD
      OUT     T4454 D3172  ; TIME.4P-RE-#5-COOLING
5490  LD      T4454
      OR      M4455  ; INREA.4P.RE.#5.UNIT.BWD
      AND     M4450  ; INREA.4P.RE.#5.AT
      ANI     M4456  ; INREA.4P.RE.#5.AT.END
      OUT     M4455  ; INREA.4P.RE.#5.UNIT.BWD
      AND     X6E9  ; 4P INFRA WELD REAR#5 CYL' BWD
      OUT     T4455 K1
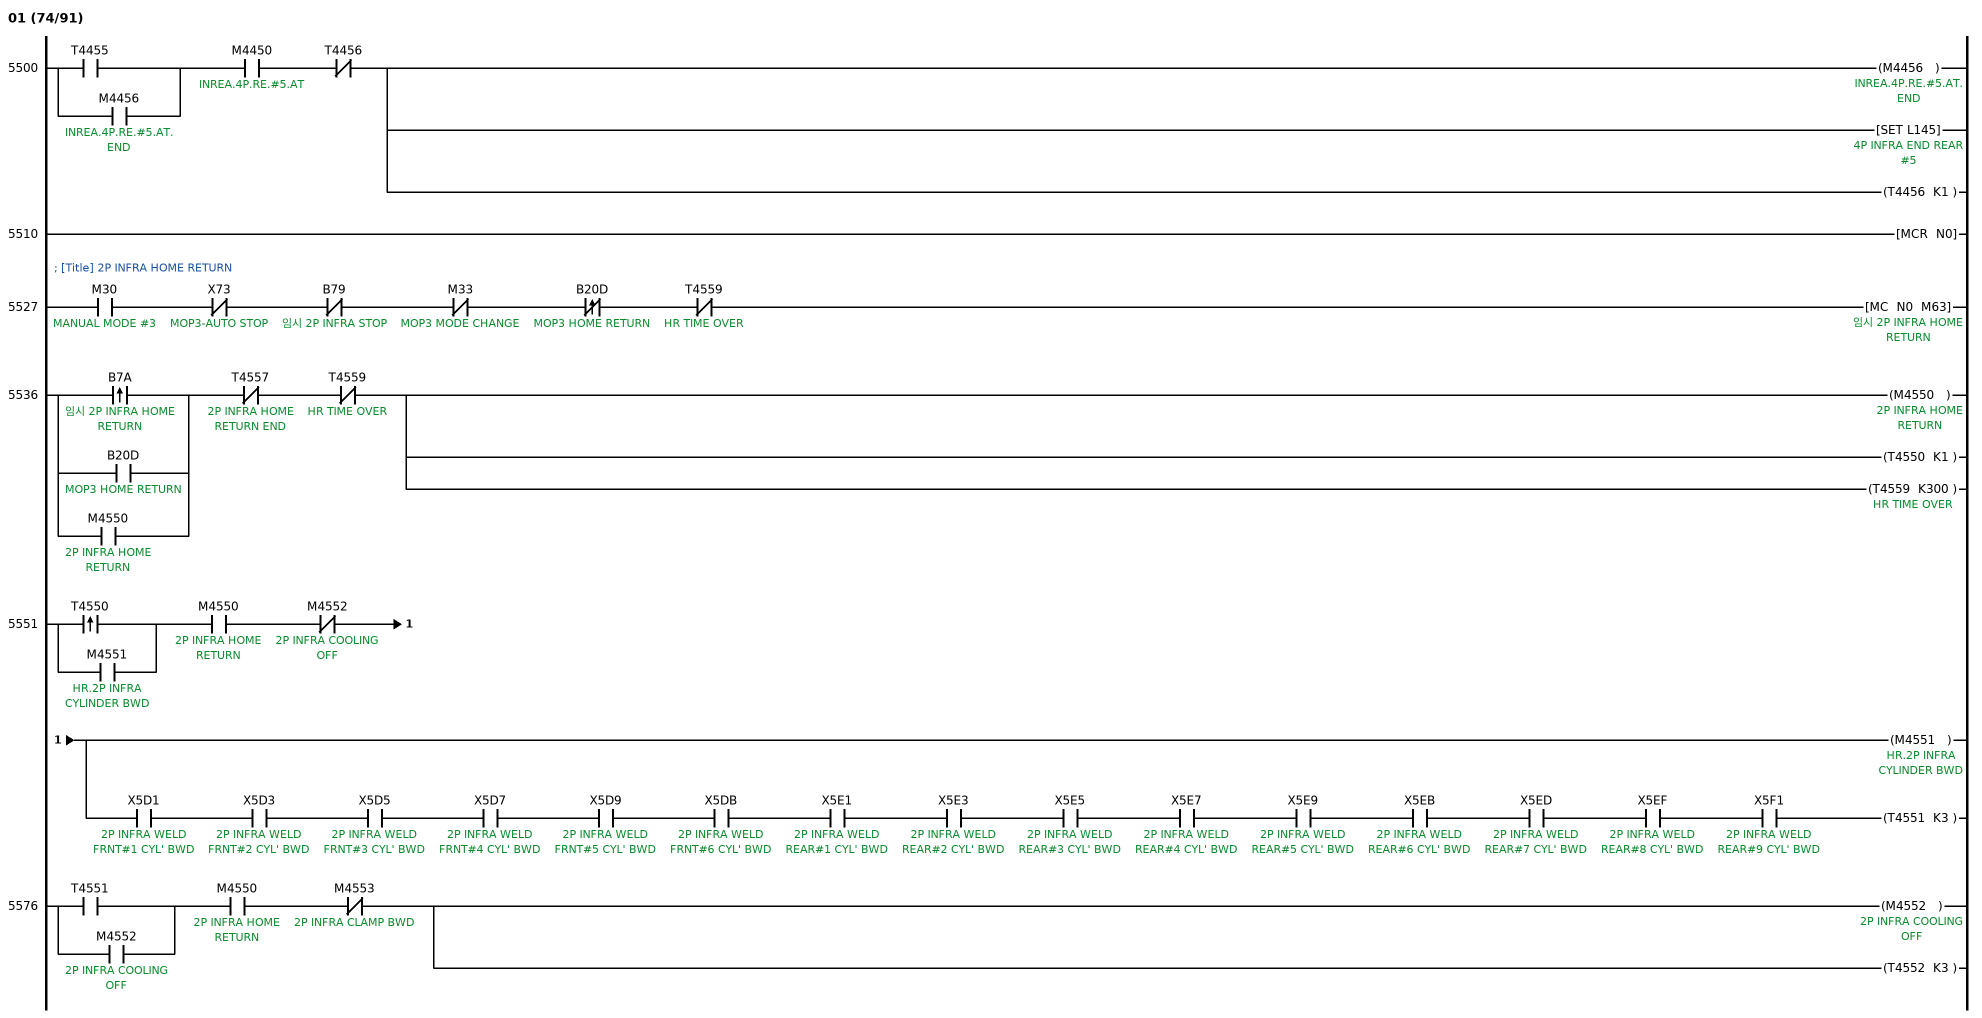
5500  LD      T4455
      OR      M4456  ; INREA.4P.RE.#5.AT.END
      AND     M4450  ; INREA.4P.RE.#5.AT
      ANI     T4456
      OUT     M4456  ; INREA.4P.RE.#5.AT.END
      SET     L145  ; 4P INFRA END REAR #5
      OUT     T4456 K1
5510  MCR     N0
; [Title] 2P INFRA HOME RETURN
5527  LD      M30  ; MANUAL MODE #3
      ANI     X73  ; MOP3-AUTO STOP
      ANI     B79  ; 임시 2P INFRA STOP
      ANI     M33  ; MOP3 MODE CHANGE
      ANDPI   B20D  ; MOP3 HOME RETURN
      ANI     T4559  ; HR TIME OVER
      MC      N0 M63  ; 임시 2P INFRA HOME RETURN
5536  LDP     B7A  ; 임시 2P INFRA HOME RETURN
      OR      B20D  ; MOP3 HOME RETURN
      OR      M4550  ; 2P INFRA HOME RETURN
      ANI     T4557  ; 2P INFRA HOME RETURN END
      ANI     T4559  ; HR TIME OVER
      OUT     M4550  ; 2P INFRA HOME RETURN
      OUT     T4550 K1
      OUT     T4559 K300  ; HR TIME OVER
5551  LDP     T4550
      OR      M4551  ; HR.2P INFRA CYLINDER BWD
      AND     M4550  ; 2P INFRA HOME RETURN
      ANI     M4552  ; 2P INFRA COOLING OFF
      OUT     M4551  ; HR.2P INFRA CYLINDER BWD
      AND     X5D1  ; 2P INFRA WELD FRNT#1 CYL' BWD
      AND     X5D3  ; 2P INFRA WELD FRNT#2 CYL' BWD
      AND     X5D5  ; 2P INFRA WELD FRNT#3 CYL' BWD
      AND     X5D7  ; 2P INFRA WELD FRNT#4 CYL' BWD
      AND     X5D9  ; 2P INFRA WELD FRNT#5 CYL' BWD
      AND     X5DB  ; 2P INFRA WELD FRNT#6 CYL' BWD
      AND     X5E1  ; 2P INFRA WELD REAR#1 CYL' BWD
      AND     X5E3  ; 2P INFRA WELD REAR#2 CYL' BWD
      AND     X5E5  ; 2P INFRA WELD REAR#3 CYL' BWD
      AND     X5E7  ; 2P INFRA WELD REAR#4 CYL' BWD
      AND     X5E9  ; 2P INFRA WELD REAR#5 CYL' BWD
      AND     X5EB  ; 2P INFRA WELD REAR#6 CYL' BWD
      AND     X5ED  ; 2P INFRA WELD REAR#7 CYL' BWD
      AND     X5EF  ; 2P INFRA WELD REAR#8 CYL' BWD
      AND     X5F1  ; 2P INFRA WELD REAR#9 CYL' BWD
      OUT     T4551 K3
5576  LD      T4551
      OR      M4552  ; 2P INFRA COOLING OFF
      AND     M4550  ; 2P INFRA HOME RETURN
      ANI     M4553  ; 2P INFRA CLAMP BWD
      OUT     M4552  ; 2P INFRA COOLING OFF
      OUT     T4552 K3
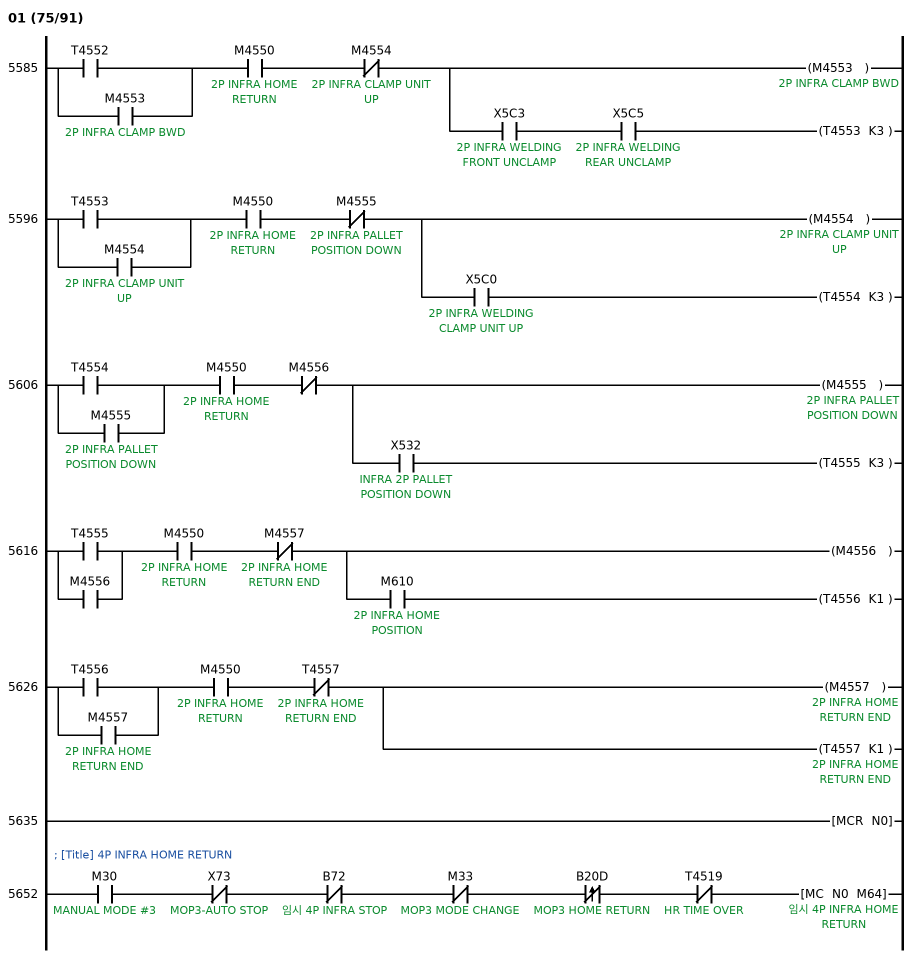
5585  LD      T4552
      OR      M4553  ; 2P INFRA CLAMP BWD
      AND     M4550  ; 2P INFRA HOME RETURN
      ANI     M4554  ; 2P INFRA CLAMP UNIT UP
      OUT     M4553  ; 2P INFRA CLAMP BWD
      AND     X5C3  ; 2P INFRA WELDING FRONT UNCLAMP
      AND     X5C5  ; 2P INFRA WELDING REAR UNCLAMP
      OUT     T4553 K3
5596  LD      T4553
      OR      M4554  ; 2P INFRA CLAMP UNIT UP
      AND     M4550  ; 2P INFRA HOME RETURN
      ANI     M4555  ; 2P INFRA PALLET POSITION DOWN
      OUT     M4554  ; 2P INFRA CLAMP UNIT UP
      AND     X5C0  ; 2P INFRA WELDING CLAMP UNIT UP
      OUT     T4554 K3
5606  LD      T4554
      OR      M4555  ; 2P INFRA PALLET POSITION DOWN
      AND     M4550  ; 2P INFRA HOME RETURN
      ANI     M4556
      OUT     M4555  ; 2P INFRA PALLET POSITION DOWN
      AND     X532  ; INFRA 2P PALLET POSITION DOWN
      OUT     T4555 K3
5616  LD      T4555
      OR      M4556
      AND     M4550  ; 2P INFRA HOME RETURN
      ANI     M4557  ; 2P INFRA HOME RETURN END
      OUT     M4556
      AND     M610  ; 2P INFRA HOME POSITION
      OUT     T4556 K1
5626  LD      T4556
      OR      M4557  ; 2P INFRA HOME RETURN END
      AND     M4550  ; 2P INFRA HOME RETURN
      ANI     T4557  ; 2P INFRA HOME RETURN END
      OUT     M4557  ; 2P INFRA HOME RETURN END
      OUT     T4557 K1  ; 2P INFRA HOME RETURN END
5635  MCR     N0
; [Title] 4P INFRA HOME RETURN
5652  LD      M30  ; MANUAL MODE #3
      ANI     X73  ; MOP3-AUTO STOP
      ANI     B72  ; 임시 4P INFRA STOP
      ANI     M33  ; MOP3 MODE CHANGE
      ANDPI   B20D  ; MOP3 HOME RETURN
      ANI     T4519  ; HR TIME OVER
      MC      N0 M64  ; 임시 4P INFRA HOME RETURN
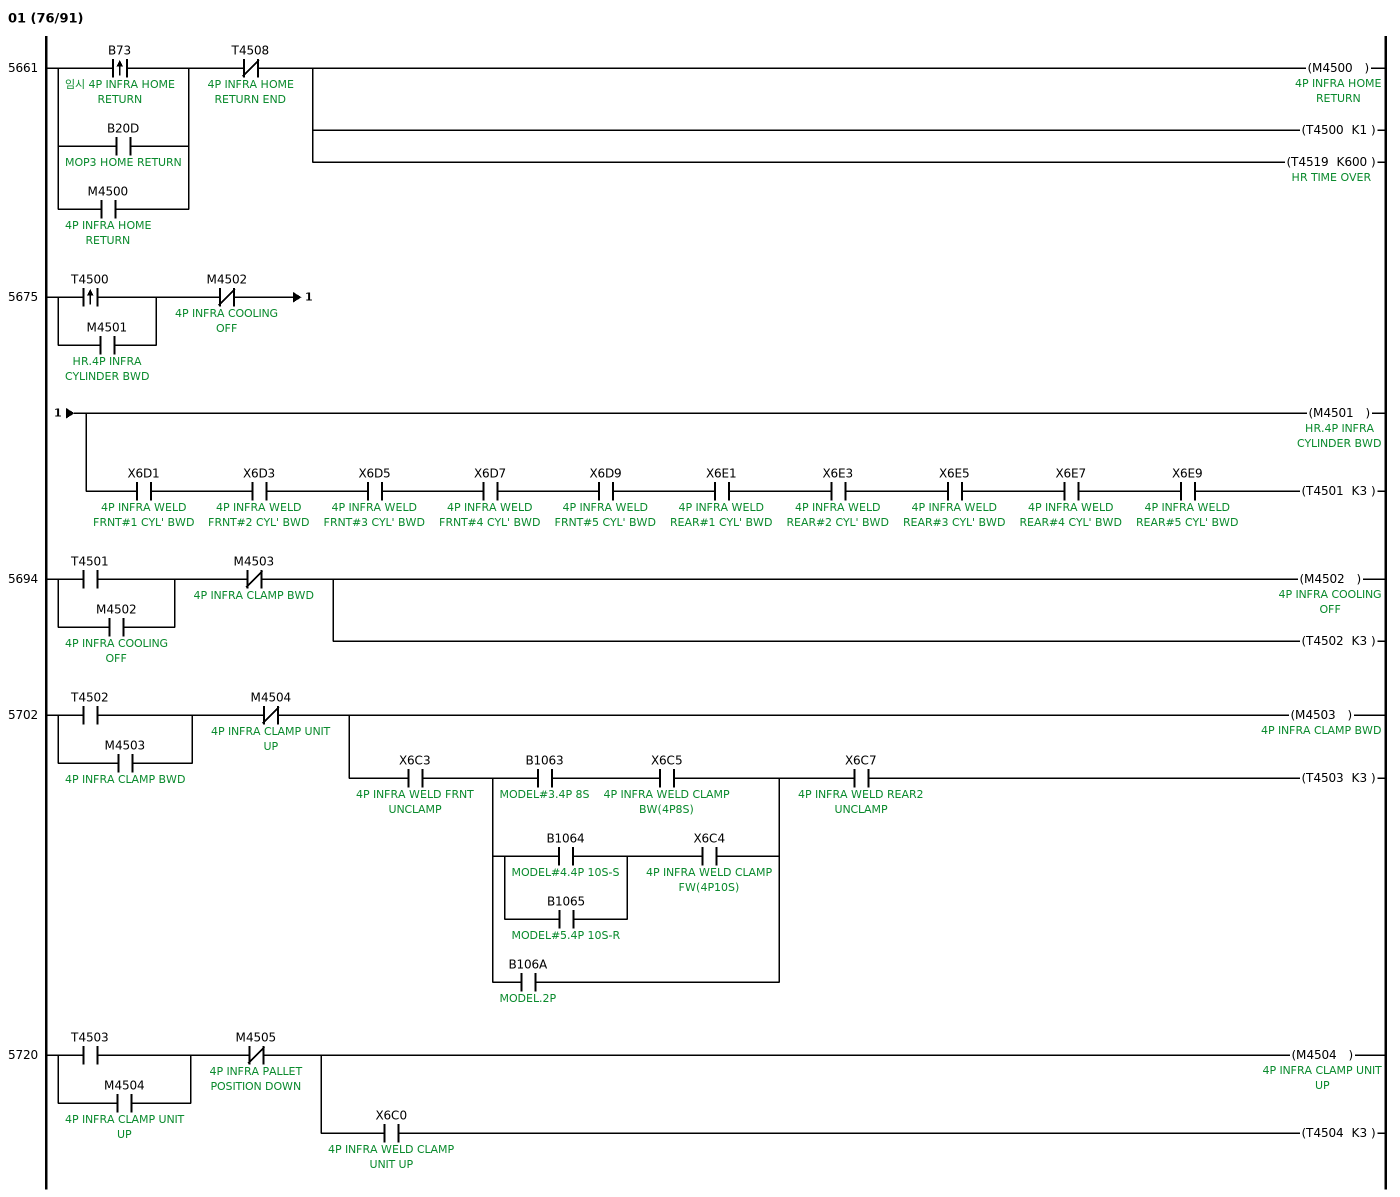
5661  LDP     B73  ; 임시 4P INFRA HOME RETURN
      OR      B20D  ; MOP3 HOME RETURN
      OR      M4500  ; 4P INFRA HOME RETURN
      ANI     T4508  ; 4P INFRA HOME RETURN END
      OUT     M4500  ; 4P INFRA HOME RETURN
      OUT     T4500 K1
      OUT     T4519 K600  ; HR TIME OVER
5675  LDP     T4500
      OR      M4501  ; HR.4P INFRA CYLINDER BWD
      ANI     M4502  ; 4P INFRA COOLING OFF
      OUT     M4501  ; HR.4P INFRA CYLINDER BWD
      AND     X6D1  ; 4P INFRA WELD FRNT#1 CYL' BWD
      AND     X6D3  ; 4P INFRA WELD FRNT#2 CYL' BWD
      AND     X6D5  ; 4P INFRA WELD FRNT#3 CYL' BWD
      AND     X6D7  ; 4P INFRA WELD FRNT#4 CYL' BWD
      AND     X6D9  ; 4P INFRA WELD FRNT#5 CYL' BWD
      AND     X6E1  ; 4P INFRA WELD REAR#1 CYL' BWD
      AND     X6E3  ; 4P INFRA WELD REAR#2 CYL' BWD
      AND     X6E5  ; 4P INFRA WELD REAR#3 CYL' BWD
      AND     X6E7  ; 4P INFRA WELD REAR#4 CYL' BWD
      AND     X6E9  ; 4P INFRA WELD REAR#5 CYL' BWD
      OUT     T4501 K3
5694  LD      T4501
      OR      M4502  ; 4P INFRA COOLING OFF
      ANI     M4503  ; 4P INFRA CLAMP BWD
      OUT     M4502  ; 4P INFRA COOLING OFF
      OUT     T4502 K3
5702  LD      T4502
      OR      M4503  ; 4P INFRA CLAMP BWD
      ANI     M4504  ; 4P INFRA CLAMP UNIT UP
      OUT     M4503  ; 4P INFRA CLAMP BWD
      AND     X6C3  ; 4P INFRA WELD FRNT UNCLAMP
      LD      B1063  ; MODEL#3.4P 8S
      AND     X6C5  ; 4P INFRA WELD CLAMP BW(4P8S)
      LD      B1064  ; MODEL#4.4P 10S-S
      OR      B1065  ; MODEL#5.4P 10S-R
      AND     X6C4  ; 4P INFRA WELD CLAMP FW(4P10S)
      ORB
      OR      B106A  ; MODEL.2P
      ANB
      AND     X6C7  ; 4P INFRA WELD REAR2 UNCLAMP
      OUT     T4503 K3
5720  LD      T4503
      OR      M4504  ; 4P INFRA CLAMP UNIT UP
      ANI     M4505  ; 4P INFRA PALLET POSITION DOWN
      OUT     M4504  ; 4P INFRA CLAMP UNIT UP
      AND     X6C0  ; 4P INFRA WELD CLAMP UNIT UP
      OUT     T4504 K3
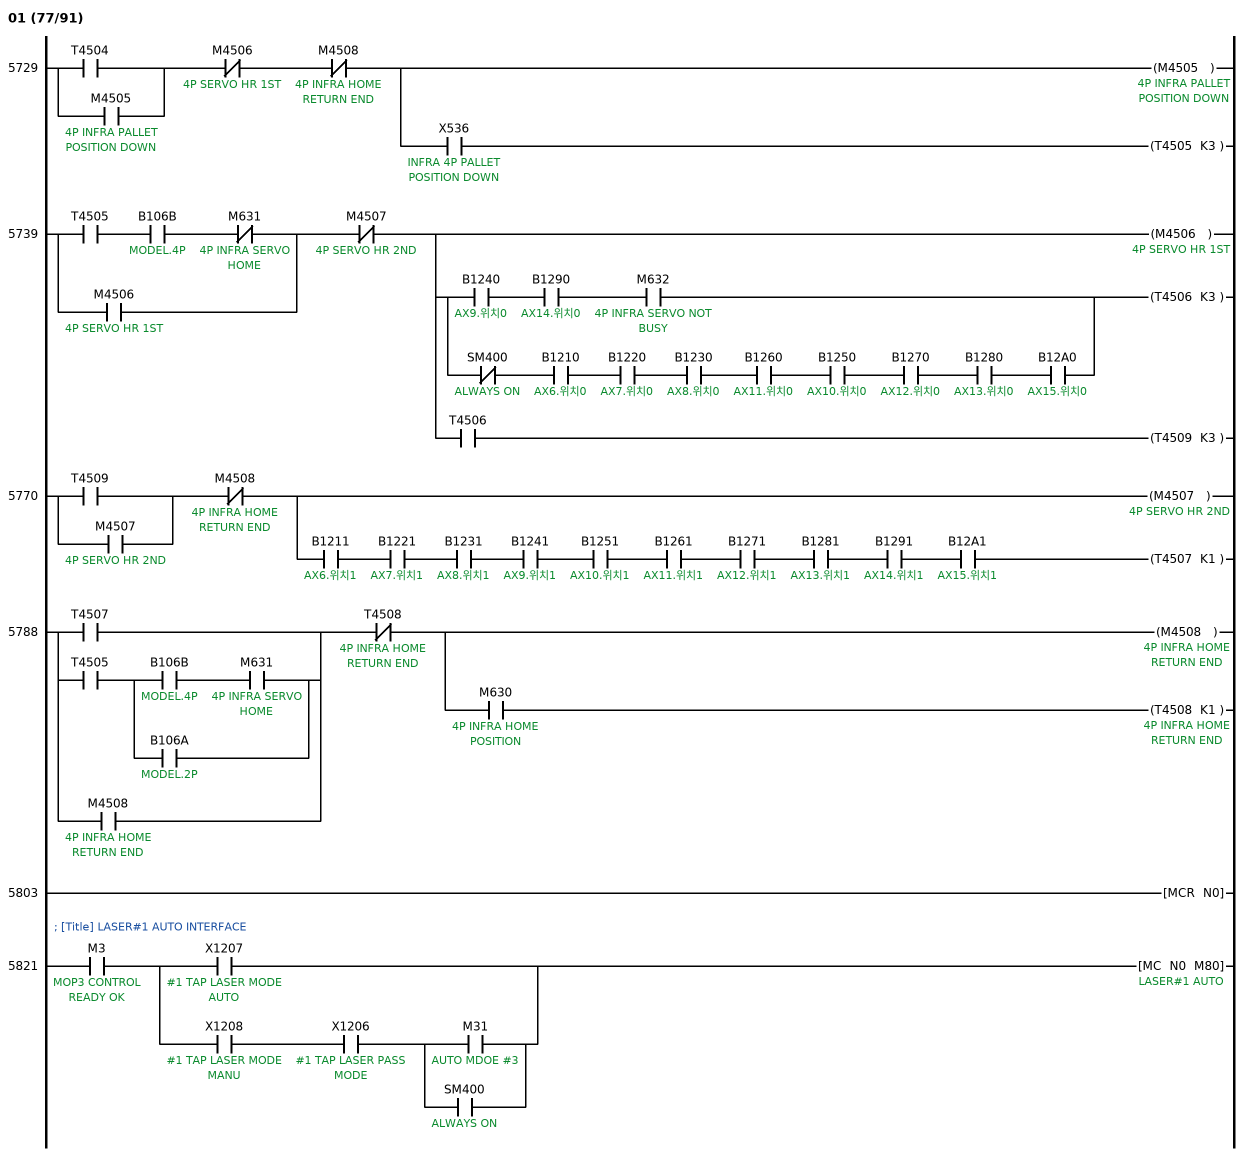
5729  LD      T4504
      OR      M4505  ; 4P INFRA PALLET POSITION DOWN
      ANI     M4506  ; 4P SERVO HR 1ST
      ANI     M4508  ; 4P INFRA HOME RETURN END
      OUT     M4505  ; 4P INFRA PALLET POSITION DOWN
      AND     X536  ; INFRA 4P PALLET POSITION DOWN
      OUT     T4505 K3
5739  LD      T4505
      AND     B106B  ; MODEL.4P
      ANI     M631  ; 4P INFRA SERVO HOME
      OR      M4506  ; 4P SERVO HR 1ST
      ANI     M4507  ; 4P SERVO HR 2ND
      OUT     M4506  ; 4P SERVO HR 1ST
      MPS
      LD      B1240  ; AX9.위치0
      AND     B1290  ; AX14.위치0
      AND     M632  ; 4P INFRA SERVO NOT BUSY
      LDI     SM400  ; ALWAYS ON
      AND     B1210  ; AX6.위치0
      AND     B1220  ; AX7.위치0
      AND     B1230  ; AX8.위치0
      AND     B1260  ; AX11.위치0
      AND     B1250  ; AX10.위치0
      AND     B1270  ; AX12.위치0
      AND     B1280  ; AX13.위치0
      AND     B12A0  ; AX15.위치0
      ORB
      ANB
      OUT     T4506 K3
      MPP
      AND     T4506
      OUT     T4509 K3
5770  LD      T4509
      OR      M4507  ; 4P SERVO HR 2ND
      ANI     M4508  ; 4P INFRA HOME RETURN END
      OUT     M4507  ; 4P SERVO HR 2ND
      AND     B1211  ; AX6.위치1
      AND     B1221  ; AX7.위치1
      AND     B1231  ; AX8.위치1
      AND     B1241  ; AX9.위치1
      AND     B1251  ; AX10.위치1
      AND     B1261  ; AX11.위치1
      AND     B1271  ; AX12.위치1
      AND     B1281  ; AX13.위치1
      AND     B1291  ; AX14.위치1
      AND     B12A1  ; AX15.위치1
      OUT     T4507 K1
5788  LD      T4507
      LD      T4505
      LD      B106B  ; MODEL.4P
      AND     M631  ; 4P INFRA SERVO HOME
      OR      B106A  ; MODEL.2P
      ANB
      ORB
      OR      M4508  ; 4P INFRA HOME RETURN END
      ANI     T4508  ; 4P INFRA HOME RETURN END
      OUT     M4508  ; 4P INFRA HOME RETURN END
      AND     M630  ; 4P INFRA HOME POSITION
      OUT     T4508 K1  ; 4P INFRA HOME RETURN END
5803  MCR     N0
; [Title] LASER#1 AUTO INTERFACE
5821  LD      M3  ; MOP3 CONTROL READY OK
      LD      X1207  ; #1 TAP LASER MODE AUTO
      LD      X1208  ; #1 TAP LASER MODE MANU
      AND     X1206  ; #1 TAP LASER PASS MODE
      LD      M31  ; AUTO MDOE #3
      OR      SM400  ; ALWAYS ON
      ANB
      ORB
      ANB
      MC      N0 M80  ; LASER#1 AUTO
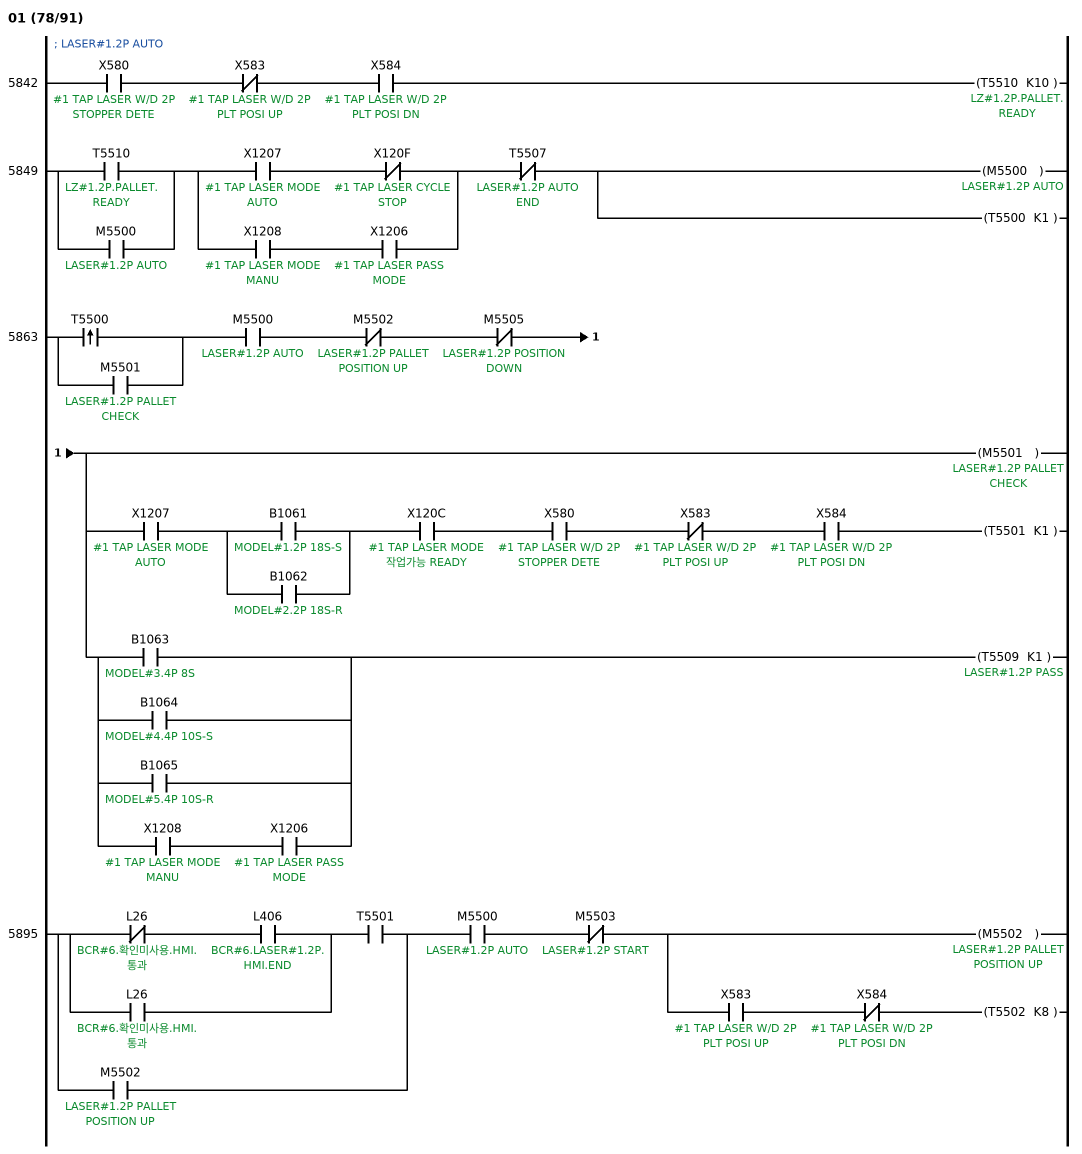
; LASER#1.2P AUTO
5842  LD      X580  ; #1 TAP LASER W/D 2P STOPPER DETE
      ANI     X583  ; #1 TAP LASER W/D 2P PLT POSI UP
      AND     X584  ; #1 TAP LASER W/D 2P PLT POSI DN
      OUT     T5510 K10  ; LZ#1.2P.PALLET.READY
5849  LD      T5510  ; LZ#1.2P.PALLET.READY
      OR      M5500  ; LASER#1.2P AUTO
      LD      X1207  ; #1 TAP LASER MODE AUTO
      ANI     X120F  ; #1 TAP LASER CYCLE STOP
      LD      X1208  ; #1 TAP LASER MODE MANU
      AND     X1206  ; #1 TAP LASER PASS MODE
      ORB
      ANB
      ANI     T5507  ; LASER#1.2P AUTO END
      OUT     M5500  ; LASER#1.2P AUTO
      OUT     T5500 K1
5863  LDP     T5500
      OR      M5501  ; LASER#1.2P PALLET CHECK
      AND     M5500  ; LASER#1.2P AUTO
      ANI     M5502  ; LASER#1.2P PALLET POSITION UP
      ANI     M5505  ; LASER#1.2P POSITION DOWN
      OUT     M5501  ; LASER#1.2P PALLET CHECK
      MPS
      AND     X1207  ; #1 TAP LASER MODE AUTO
      LD      B1061  ; MODEL#1.2P 18S-S
      OR      B1062  ; MODEL#2.2P 18S-R
      ANB
      AND     X120C  ; #1 TAP LASER MODE 작업가능 READY
      AND     X580  ; #1 TAP LASER W/D 2P STOPPER DETE
      ANI     X583  ; #1 TAP LASER W/D 2P PLT POSI UP
      AND     X584  ; #1 TAP LASER W/D 2P PLT POSI DN
      OUT     T5501 K1
      MPP
      LD      B1063  ; MODEL#3.4P 8S
      OR      B1064  ; MODEL#4.4P 10S-S
      OR      B1065  ; MODEL#5.4P 10S-R
      LD      X1208  ; #1 TAP LASER MODE MANU
      AND     X1206  ; #1 TAP LASER PASS MODE
      ORB
      ANB
      OUT     T5509 K1  ; LASER#1.2P PASS
5895  LDI     L26  ; BCR#6.확인미사용.HMI.통과
      AND     L406  ; BCR#6.LASER#1.2P.HMI.END
      OR      L26  ; BCR#6.확인미사용.HMI.통과
      AND     T5501
      OR      M5502  ; LASER#1.2P PALLET POSITION UP
      AND     M5500  ; LASER#1.2P AUTO
      ANI     M5503  ; LASER#1.2P START
      OUT     M5502  ; LASER#1.2P PALLET POSITION UP
      AND     X583  ; #1 TAP LASER W/D 2P PLT POSI UP
      ANI     X584  ; #1 TAP LASER W/D 2P PLT POSI DN
      OUT     T5502 K8
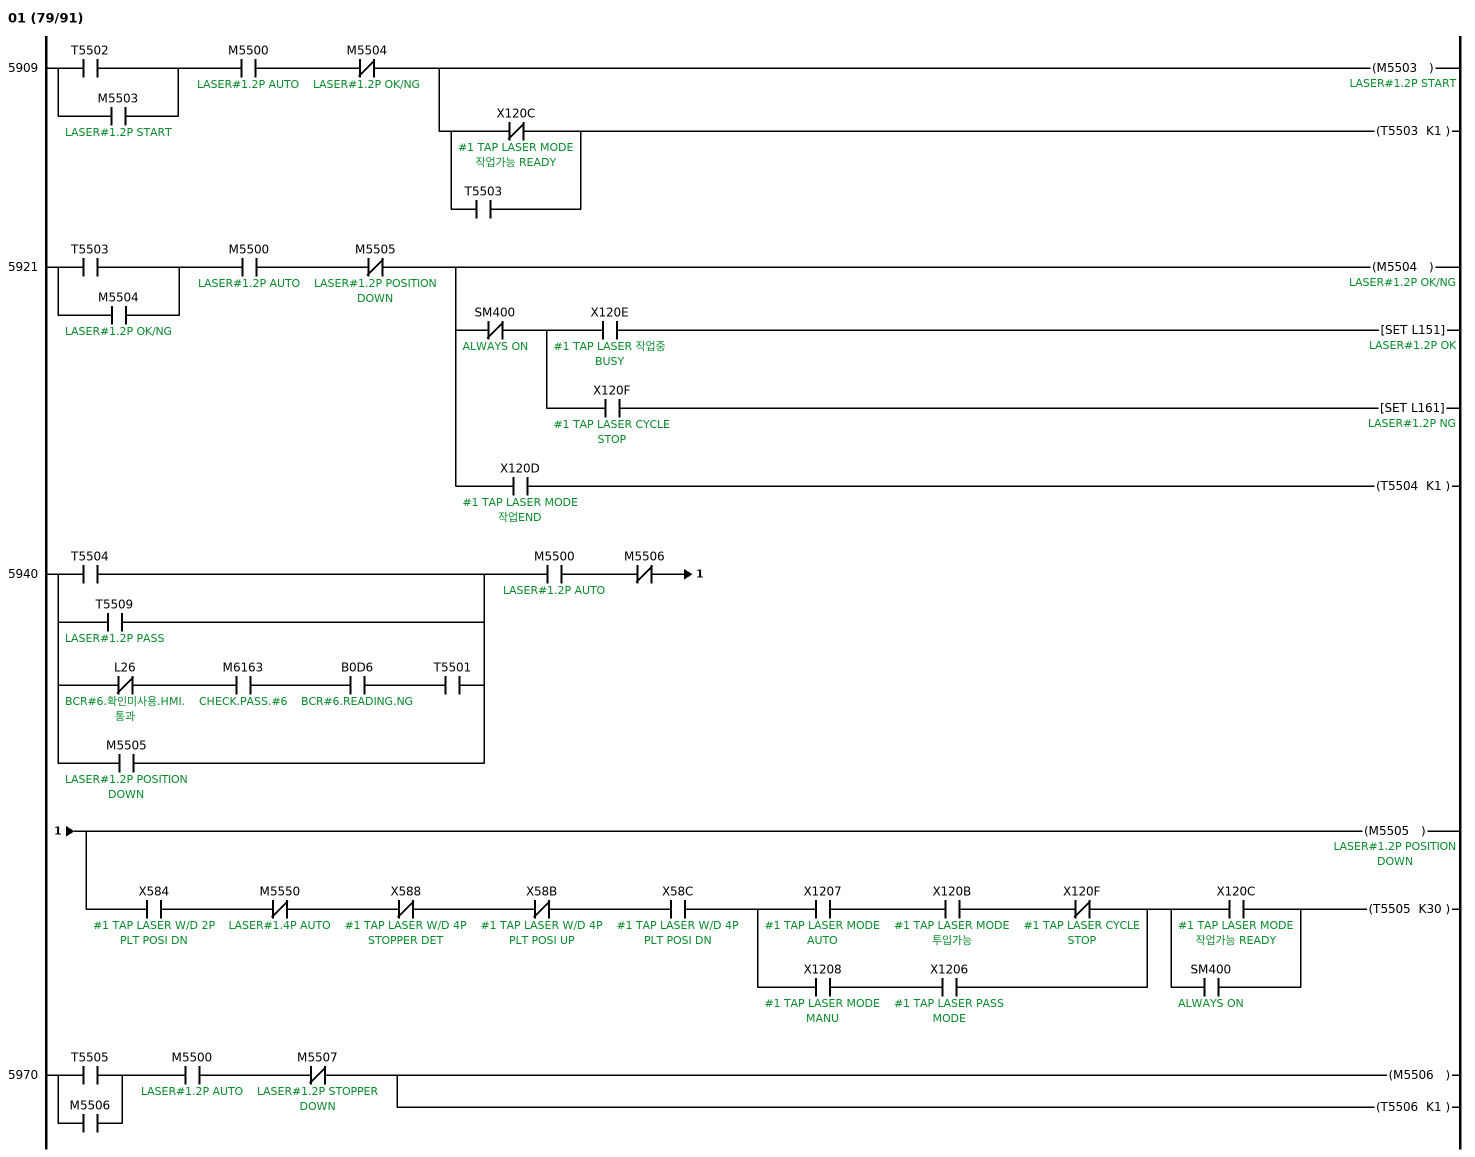
5909  LD      T5502
      OR      M5503  ; LASER#1.2P START
      AND     M5500  ; LASER#1.2P AUTO
      ANI     M5504  ; LASER#1.2P OK/NG
      OUT     M5503  ; LASER#1.2P START
      LDI     X120C  ; #1 TAP LASER MODE 작업가능 READY
      OR      T5503
      ANB
      OUT     T5503 K1
5921  LD      T5503
      OR      M5504  ; LASER#1.2P OK/NG
      AND     M5500  ; LASER#1.2P AUTO
      ANI     M5505  ; LASER#1.2P POSITION DOWN
      OUT     M5504  ; LASER#1.2P OK/NG
      MPS
      ANI     SM400  ; ALWAYS ON
      MPS
      AND     X120E  ; #1 TAP LASER 작업중 BUSY
      SET     L151  ; LASER#1.2P OK
      MPP
      AND     X120F  ; #1 TAP LASER CYCLE STOP
      SET     L161  ; LASER#1.2P NG
      MPP
      AND     X120D  ; #1 TAP LASER MODE 작업END
      OUT     T5504 K1
5940  LD      T5504
      OR      T5509  ; LASER#1.2P PASS
      LDI     L26  ; BCR#6.확인미사용.HMI.통과
      AND     M6163  ; CHECK.PASS.#6
      AND     B0D6  ; BCR#6.READING.NG
      AND     T5501
      ORB
      OR      M5505  ; LASER#1.2P POSITION DOWN
      AND     M5500  ; LASER#1.2P AUTO
      ANI     M5506
      OUT     M5505  ; LASER#1.2P POSITION DOWN
      AND     X584  ; #1 TAP LASER W/D 2P PLT POSI DN
      ANI     M5550  ; LASER#1.4P AUTO
      ANI     X588  ; #1 TAP LASER W/D 4P STOPPER DET
      ANI     X58B  ; #1 TAP LASER W/D 4P PLT POSI UP
      AND     X58C  ; #1 TAP LASER W/D 4P PLT POSI DN
      LD      X1207  ; #1 TAP LASER MODE AUTO
      AND     X120B  ; #1 TAP LASER MODE 투입가능
      ANI     X120F  ; #1 TAP LASER CYCLE STOP
      LD      X1208  ; #1 TAP LASER MODE MANU
      AND     X1206  ; #1 TAP LASER PASS MODE
      ORB
      ANB
      LD      X120C  ; #1 TAP LASER MODE 작업가능 READY
      OR      SM400  ; ALWAYS ON
      ANB
      OUT     T5505 K30
5970  LD      T5505
      OR      M5506
      AND     M5500  ; LASER#1.2P AUTO
      ANI     M5507  ; LASER#1.2P STOPPER DOWN
      OUT     M5506
      OUT     T5506 K1
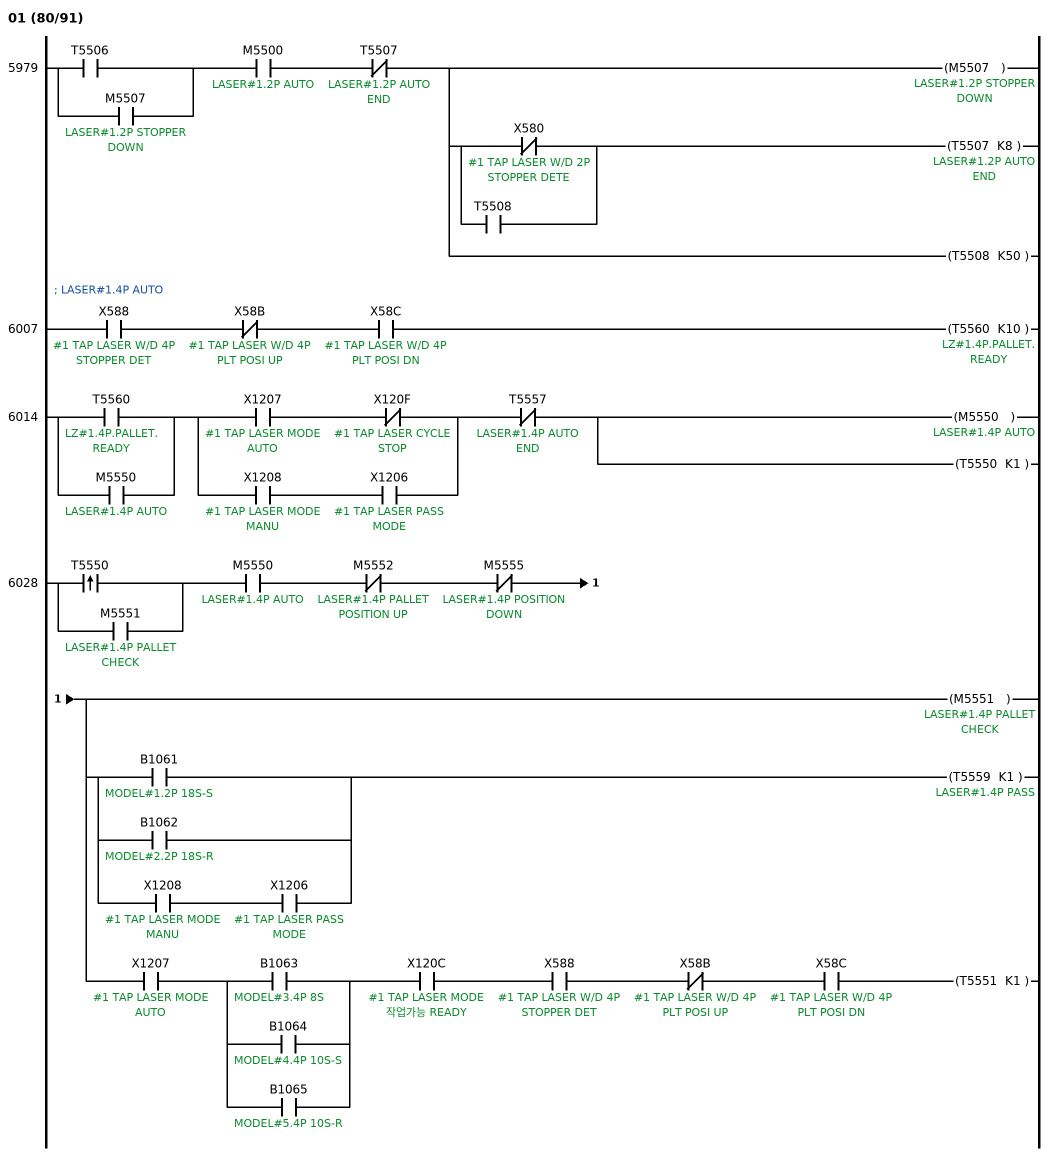
5979  LD      T5506
      OR      M5507  ; LASER#1.2P STOPPER DOWN
      AND     M5500  ; LASER#1.2P AUTO
      ANI     T5507  ; LASER#1.2P AUTO END
      OUT     M5507  ; LASER#1.2P STOPPER DOWN
      MPS
      LDI     X580  ; #1 TAP LASER W/D 2P STOPPER DETE
      OR      T5508
      ANB
      OUT     T5507 K8  ; LASER#1.2P AUTO END
      MPP
      OUT     T5508 K50
; LASER#1.4P AUTO
6007  LD      X588  ; #1 TAP LASER W/D 4P STOPPER DET
      ANI     X58B  ; #1 TAP LASER W/D 4P PLT POSI UP
      AND     X58C  ; #1 TAP LASER W/D 4P PLT POSI DN
      OUT     T5560 K10  ; LZ#1.4P.PALLET.READY
6014  LD      T5560  ; LZ#1.4P.PALLET.READY
      OR      M5550  ; LASER#1.4P AUTO
      LD      X1207  ; #1 TAP LASER MODE AUTO
      ANI     X120F  ; #1 TAP LASER CYCLE STOP
      LD      X1208  ; #1 TAP LASER MODE MANU
      AND     X1206  ; #1 TAP LASER PASS MODE
      ORB
      ANB
      ANI     T5557  ; LASER#1.4P AUTO END
      OUT     M5550  ; LASER#1.4P AUTO
      OUT     T5550 K1
6028  LDP     T5550
      OR      M5551  ; LASER#1.4P PALLET CHECK
      AND     M5550  ; LASER#1.4P AUTO
      ANI     M5552  ; LASER#1.4P PALLET POSITION UP
      ANI     M5555  ; LASER#1.4P POSITION DOWN
      OUT     M5551  ; LASER#1.4P PALLET CHECK
      MPS
      LD      B1061  ; MODEL#1.2P 18S-S
      OR      B1062  ; MODEL#2.2P 18S-R
      LD      X1208  ; #1 TAP LASER MODE MANU
      AND     X1206  ; #1 TAP LASER PASS MODE
      ORB
      ANB
      OUT     T5559 K1  ; LASER#1.4P PASS
      MPP
      AND     X1207  ; #1 TAP LASER MODE AUTO
      LD      B1063  ; MODEL#3.4P 8S
      OR      B1064  ; MODEL#4.4P 10S-S
      OR      B1065  ; MODEL#5.4P 10S-R
      ANB
      AND     X120C  ; #1 TAP LASER MODE 작업가능 READY
      AND     X588  ; #1 TAP LASER W/D 4P STOPPER DET
      ANI     X58B  ; #1 TAP LASER W/D 4P PLT POSI UP
      AND     X58C  ; #1 TAP LASER W/D 4P PLT POSI DN
      OUT     T5551 K1
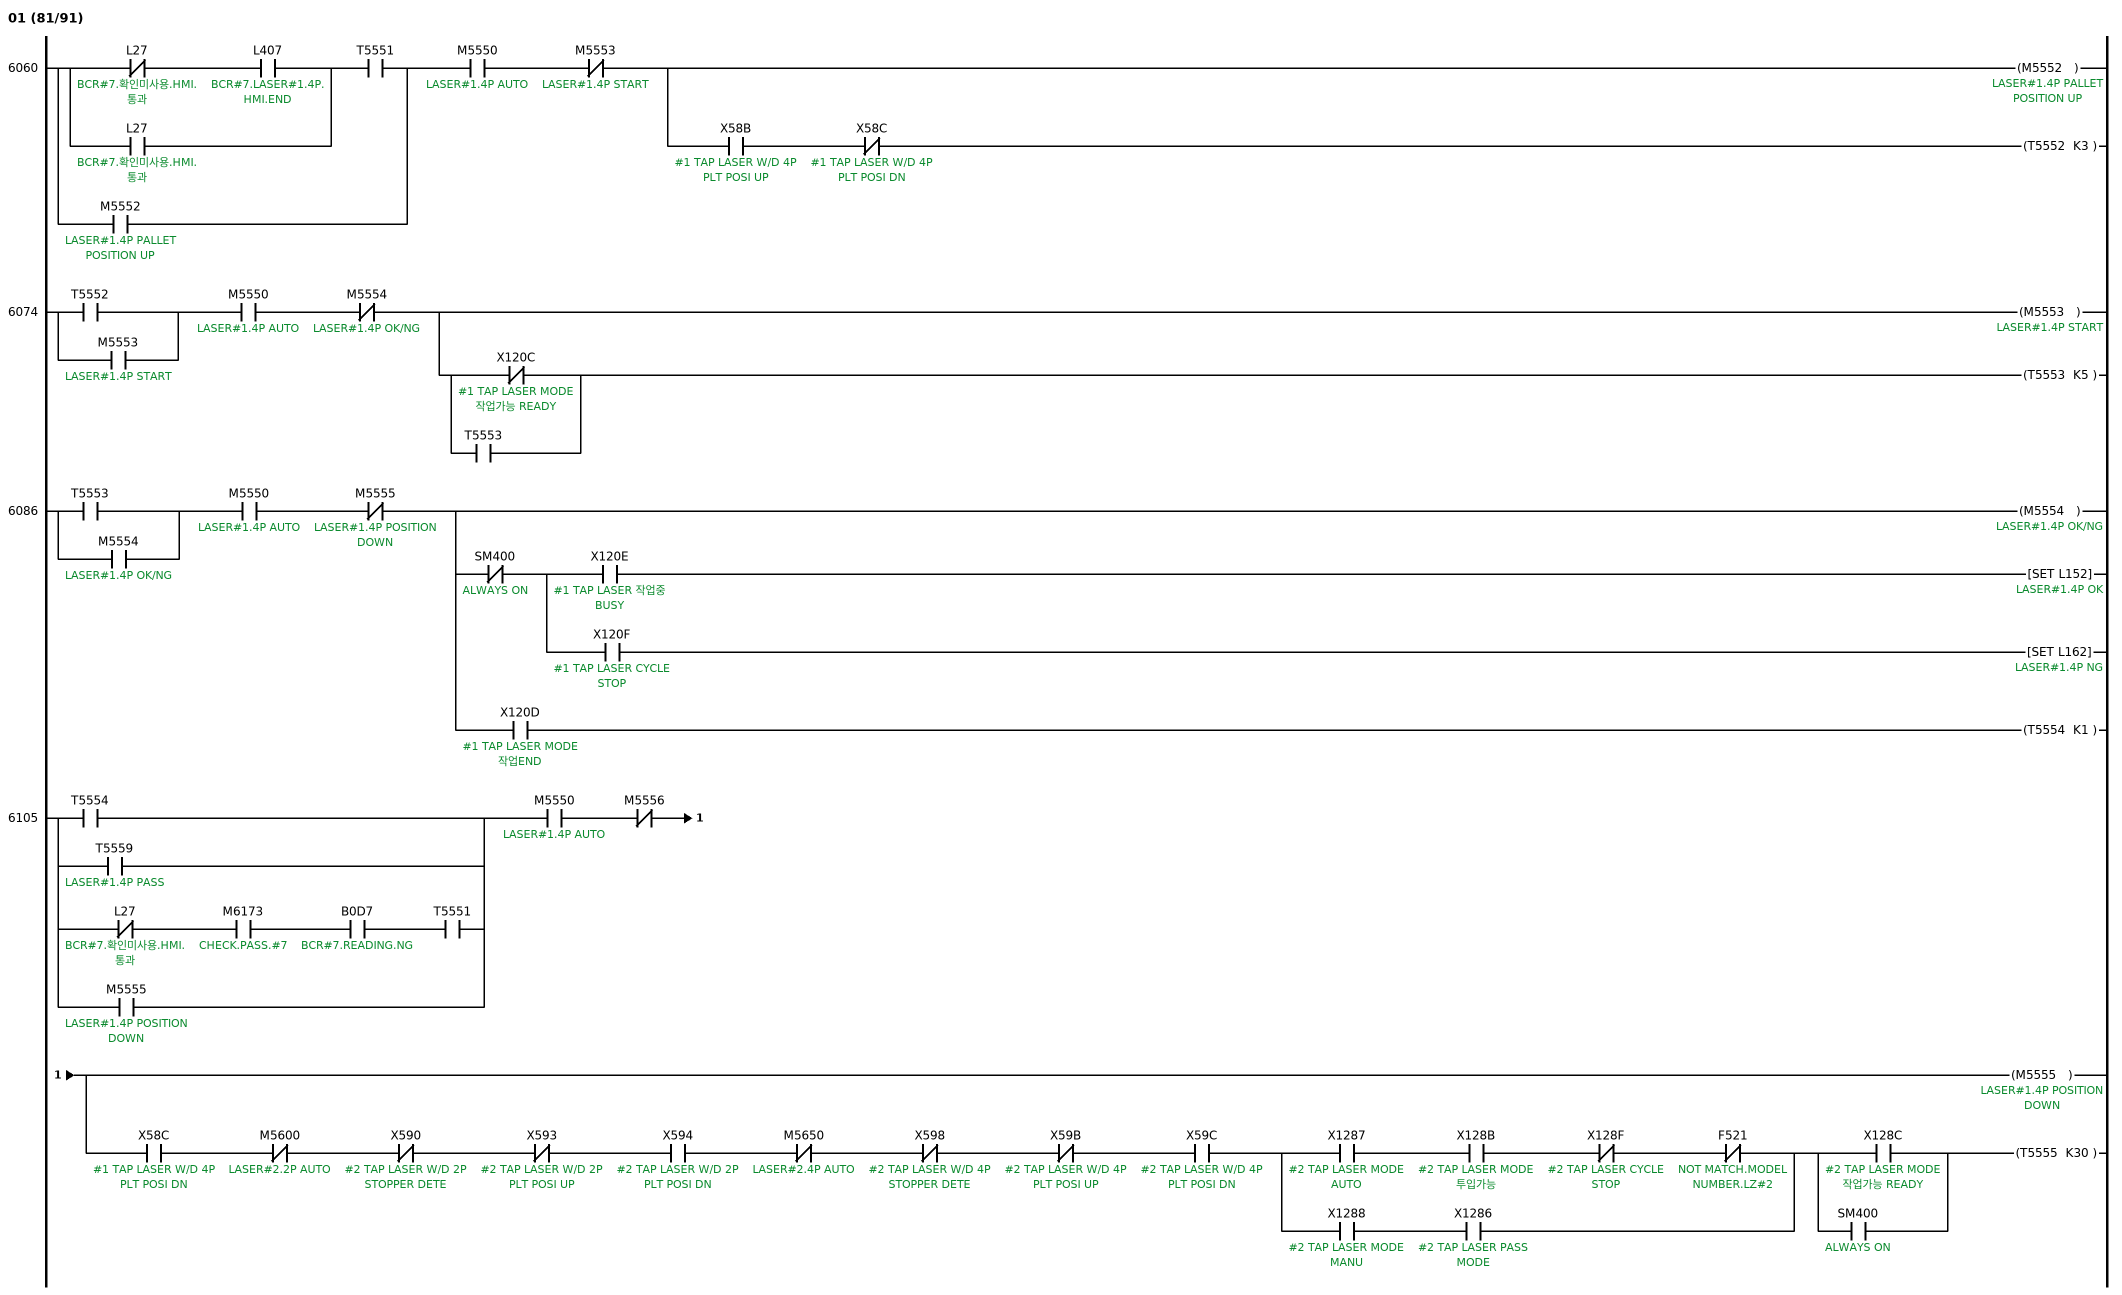
6060  LDI     L27  ; BCR#7.확인미사용.HMI.통과
      AND     L407  ; BCR#7.LASER#1.4P.HMI.END
      OR      L27  ; BCR#7.확인미사용.HMI.통과
      AND     T5551
      OR      M5552  ; LASER#1.4P PALLET POSITION UP
      AND     M5550  ; LASER#1.4P AUTO
      ANI     M5553  ; LASER#1.4P START
      OUT     M5552  ; LASER#1.4P PALLET POSITION UP
      AND     X58B  ; #1 TAP LASER W/D 4P PLT POSI UP
      ANI     X58C  ; #1 TAP LASER W/D 4P PLT POSI DN
      OUT     T5552 K3
6074  LD      T5552
      OR      M5553  ; LASER#1.4P START
      AND     M5550  ; LASER#1.4P AUTO
      ANI     M5554  ; LASER#1.4P OK/NG
      OUT     M5553  ; LASER#1.4P START
      LDI     X120C  ; #1 TAP LASER MODE 작업가능 READY
      OR      T5553
      ANB
      OUT     T5553 K5
6086  LD      T5553
      OR      M5554  ; LASER#1.4P OK/NG
      AND     M5550  ; LASER#1.4P AUTO
      ANI     M5555  ; LASER#1.4P POSITION DOWN
      OUT     M5554  ; LASER#1.4P OK/NG
      MPS
      ANI     SM400  ; ALWAYS ON
      MPS
      AND     X120E  ; #1 TAP LASER 작업중 BUSY
      SET     L152  ; LASER#1.4P OK
      MPP
      AND     X120F  ; #1 TAP LASER CYCLE STOP
      SET     L162  ; LASER#1.4P NG
      MPP
      AND     X120D  ; #1 TAP LASER MODE 작업END
      OUT     T5554 K1
6105  LD      T5554
      OR      T5559  ; LASER#1.4P PASS
      LDI     L27  ; BCR#7.확인미사용.HMI.통과
      AND     M6173  ; CHECK.PASS.#7
      AND     B0D7  ; BCR#7.READING.NG
      AND     T5551
      ORB
      OR      M5555  ; LASER#1.4P POSITION DOWN
      AND     M5550  ; LASER#1.4P AUTO
      ANI     M5556
      OUT     M5555  ; LASER#1.4P POSITION DOWN
      AND     X58C  ; #1 TAP LASER W/D 4P PLT POSI DN
      ANI     M5600  ; LASER#2.2P AUTO
      ANI     X590  ; #2 TAP LASER W/D 2P STOPPER DETE
      ANI     X593  ; #2 TAP LASER W/D 2P PLT POSI UP
      AND     X594  ; #2 TAP LASER W/D 2P PLT POSI DN
      ANI     M5650  ; LASER#2.4P AUTO
      ANI     X598  ; #2 TAP LASER W/D 4P STOPPER DETE
      ANI     X59B  ; #2 TAP LASER W/D 4P PLT POSI UP
      AND     X59C  ; #2 TAP LASER W/D 4P PLT POSI DN
      LD      X1287  ; #2 TAP LASER MODE AUTO
      AND     X128B  ; #2 TAP LASER MODE 투입가능
      ANI     X128F  ; #2 TAP LASER CYCLE STOP
      ANI     F521  ; NOT MATCH.MODEL NUMBER.LZ#2
      LD      X1288  ; #2 TAP LASER MODE MANU
      AND     X1286  ; #2 TAP LASER PASS MODE
      ORB
      ANB
      LD      X128C  ; #2 TAP LASER MODE 작업가능 READY
      OR      SM400  ; ALWAYS ON
      ANB
      OUT     T5555 K30
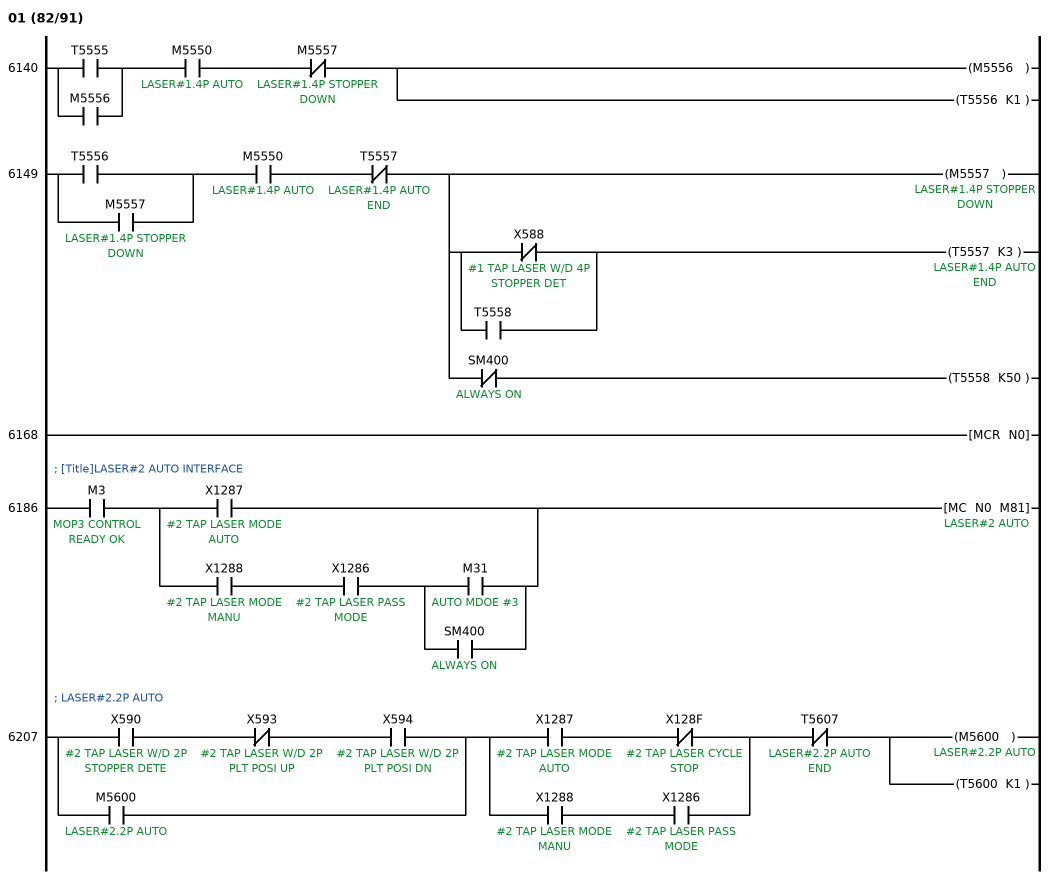
6140  LD      T5555
      OR      M5556
      AND     M5550  ; LASER#1.4P AUTO
      ANI     M5557  ; LASER#1.4P STOPPER DOWN
      OUT     M5556
      OUT     T5556 K1
6149  LD      T5556
      OR      M5557  ; LASER#1.4P STOPPER DOWN
      AND     M5550  ; LASER#1.4P AUTO
      ANI     T5557  ; LASER#1.4P AUTO END
      OUT     M5557  ; LASER#1.4P STOPPER DOWN
      MPS
      LDI     X588  ; #1 TAP LASER W/D 4P STOPPER DET
      OR      T5558
      ANB
      OUT     T5557 K3  ; LASER#1.4P AUTO END
      MPP
      ANI     SM400  ; ALWAYS ON
      OUT     T5558 K50
6168  MCR     N0
; [Title]LASER#2 AUTO INTERFACE
6186  LD      M3  ; MOP3 CONTROL READY OK
      LD      X1287  ; #2 TAP LASER MODE AUTO
      LD      X1288  ; #2 TAP LASER MODE MANU
      AND     X1286  ; #2 TAP LASER PASS MODE
      LD      M31  ; AUTO MDOE #3
      OR      SM400  ; ALWAYS ON
      ANB
      ORB
      ANB
      MC      N0 M81  ; LASER#2 AUTO
; LASER#2.2P AUTO
6207  LD      X590  ; #2 TAP LASER W/D 2P STOPPER DETE
      ANI     X593  ; #2 TAP LASER W/D 2P PLT POSI UP
      AND     X594  ; #2 TAP LASER W/D 2P PLT POSI DN
      OR      M5600  ; LASER#2.2P AUTO
      LD      X1287  ; #2 TAP LASER MODE AUTO
      ANI     X128F  ; #2 TAP LASER CYCLE STOP
      LD      X1288  ; #2 TAP LASER MODE MANU
      AND     X1286  ; #2 TAP LASER PASS MODE
      ORB
      ANB
      ANI     T5607  ; LASER#2.2P AUTO END
      OUT     M5600  ; LASER#2.2P AUTO
      OUT     T5600 K1
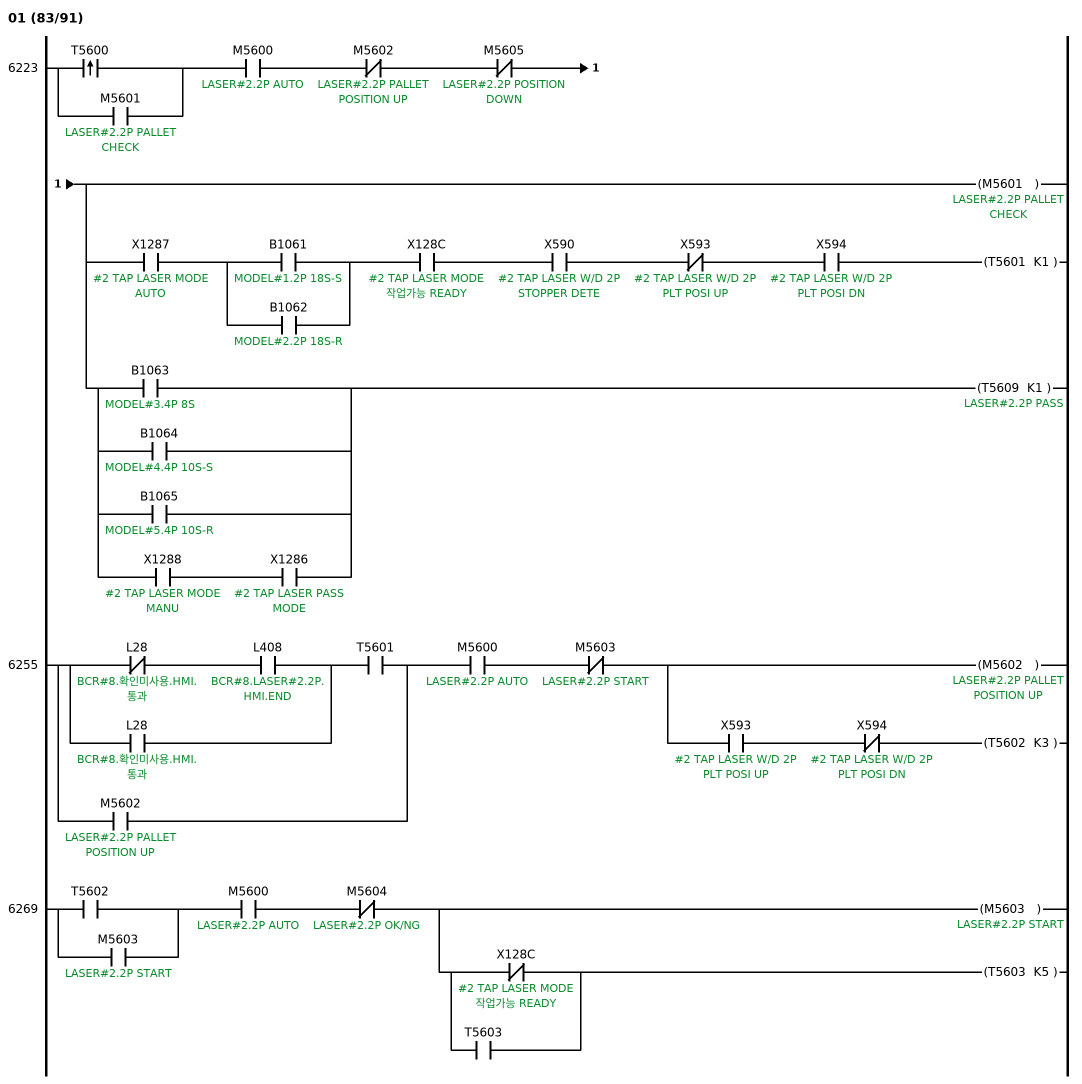
6223  LDP     T5600
      OR      M5601  ; LASER#2.2P PALLET CHECK
      AND     M5600  ; LASER#2.2P AUTO
      ANI     M5602  ; LASER#2.2P PALLET POSITION UP
      ANI     M5605  ; LASER#2.2P POSITION DOWN
      OUT     M5601  ; LASER#2.2P PALLET CHECK
      MPS
      AND     X1287  ; #2 TAP LASER MODE AUTO
      LD      B1061  ; MODEL#1.2P 18S-S
      OR      B1062  ; MODEL#2.2P 18S-R
      ANB
      AND     X128C  ; #2 TAP LASER MODE 작업가능 READY
      AND     X590  ; #2 TAP LASER W/D 2P STOPPER DETE
      ANI     X593  ; #2 TAP LASER W/D 2P PLT POSI UP
      AND     X594  ; #2 TAP LASER W/D 2P PLT POSI DN
      OUT     T5601 K1
      MPP
      LD      B1063  ; MODEL#3.4P 8S
      OR      B1064  ; MODEL#4.4P 10S-S
      OR      B1065  ; MODEL#5.4P 10S-R
      LD      X1288  ; #2 TAP LASER MODE MANU
      AND     X1286  ; #2 TAP LASER PASS MODE
      ORB
      ANB
      OUT     T5609 K1  ; LASER#2.2P PASS
6255  LDI     L28  ; BCR#8.확인미사용.HMI.통과
      AND     L408  ; BCR#8.LASER#2.2P.HMI.END
      OR      L28  ; BCR#8.확인미사용.HMI.통과
      AND     T5601
      OR      M5602  ; LASER#2.2P PALLET POSITION UP
      AND     M5600  ; LASER#2.2P AUTO
      ANI     M5603  ; LASER#2.2P START
      OUT     M5602  ; LASER#2.2P PALLET POSITION UP
      AND     X593  ; #2 TAP LASER W/D 2P PLT POSI UP
      ANI     X594  ; #2 TAP LASER W/D 2P PLT POSI DN
      OUT     T5602 K3
6269  LD      T5602
      OR      M5603  ; LASER#2.2P START
      AND     M5600  ; LASER#2.2P AUTO
      ANI     M5604  ; LASER#2.2P OK/NG
      OUT     M5603  ; LASER#2.2P START
      LDI     X128C  ; #2 TAP LASER MODE 작업가능 READY
      OR      T5603
      ANB
      OUT     T5603 K5
